  PROC DrawPart13()
    MoveL Offs(pOrigin,108.13,133.18,0.00),v40,z0,tPen\WObj:=wPaper;
    MoveL Offs(pOrigin,107.17,132.22,0.00),v40,z0,tPen\WObj:=wPaper;
    MoveL Offs(pOrigin,106.24,132.34,0.00),v40,z0,tPen\WObj:=wPaper;
    MoveL Offs(pOrigin,132.55,106.03,0.00),v40,z0,tPen\WObj:=wPaper;
    MoveL Offs(pOrigin,132.03,106.30,0.00),v40,z0,tPen\WObj:=wPaper;
    MoveL Offs(pOrigin,118.67,92.94,0.00),v40,z0,tPen\WObj:=wPaper;
    MoveL Offs(pOrigin,118.15,92.06,0.00),v40,z0,tPen\WObj:=wPaper;
    MoveL Offs(pOrigin,106.16,104.04,0.00),v40,z0,tPen\WObj:=wPaper;
    MoveL Offs(pOrigin,106.93,103.61,0.00),v40,z0,tPen\WObj:=wPaper;
    MoveL Offs(pOrigin,132.39,129.07,0.00),v40,z0,tPen\WObj:=wPaper;
    MoveL Offs(pOrigin,131.45,128.70,0.00),v40,z0,tPen\WObj:=wPaper;
    MoveL Offs(pOrigin,107.90,128.70,0.00),v40,z0,tPen\WObj:=wPaper;
    MoveL Offs(pOrigin,106.97,129.03,0.00),v40,z0,tPen\WObj:=wPaper;
    MoveL Offs(pOrigin,111.11,133.17,0.00),v40,fine,tPen\WObj:=wPaper;
    MoveL Offs(pOrigin,111.11,133.17,6.00),v60,z5,tPen\WObj:=wPaper;
    MoveL Offs(pOrigin,110.40,134.16,6.00),vTravel,z5,tPen\WObj:=wPaper;
    MoveL Offs(pOrigin,110.40,134.16,0.00),v60,z0,tPen\WObj:=wPaper;
    MoveL Offs(pOrigin,132.46,112.10,0.00),v40,z0,tPen\WObj:=wPaper;
    MoveL Offs(pOrigin,131.80,112.05,0.00),v40,z0,tPen\WObj:=wPaper;
    MoveL Offs(pOrigin,112.71,92.96,0.00),v40,z0,tPen\WObj:=wPaper;
    MoveL Offs(pOrigin,112.30,91.93,0.00),v40,z0,tPen\WObj:=wPaper;
    MoveL Offs(pOrigin,106.25,97.98,0.00),v40,z0,tPen\WObj:=wPaper;
    MoveL Offs(pOrigin,106.95,97.65,0.00),v40,z0,tPen\WObj:=wPaper;
    MoveL Offs(pOrigin,132.20,122.90,0.00),v40,z0,tPen\WObj:=wPaper;
    MoveL Offs(pOrigin,131.30,123.42,0.00),v40,z0,tPen\WObj:=wPaper;
    MoveL Offs(pOrigin,107.90,123.42,0.00),v40,z0,tPen\WObj:=wPaper;
    MoveL Offs(pOrigin,107.90,124.47,0.00),v40,z0,tPen\WObj:=wPaper;
    MoveL Offs(pOrigin,131.30,124.47,0.00),v40,z0,tPen\WObj:=wPaper;
    MoveL Offs(pOrigin,132.09,124.28,0.00),v40,z0,tPen\WObj:=wPaper;
    MoveL Offs(pOrigin,106.95,99.14,0.00),v40,z0,tPen\WObj:=wPaper;
    MoveL Offs(pOrigin,107.75,99.13,0.00),v40,z0,tPen\WObj:=wPaper;
    MoveL Offs(pOrigin,131.45,99.13,0.00),v40,z0,tPen\WObj:=wPaper;
    MoveL Offs(pOrigin,132.05,98.86,0.00),v40,z0,tPen\WObj:=wPaper;
    MoveL Offs(pOrigin,126.32,93.13,0.00),v40,z0,tPen\WObj:=wPaper;
    MoveL Offs(pOrigin,126.87,92.30,0.00),v40,z0,tPen\WObj:=wPaper;
    MoveL Offs(pOrigin,106.08,113.08,0.00),v40,z0,tPen\WObj:=wPaper;
    MoveL Offs(pOrigin,106.91,112.55,0.00),v40,z0,tPen\WObj:=wPaper;
    MoveL Offs(pOrigin,127.70,133.33,0.00),v40,z0,tPen\WObj:=wPaper;
    MoveL Offs(pOrigin,126.99,133.99,0.00),v40,z0,tPen\WObj:=wPaper;
    MoveL Offs(pOrigin,155.31,105.67,0.00),v40,z0,tPen\WObj:=wPaper;
    MoveL Offs(pOrigin,155.95,106.53,0.00),v40,z0,tPen\WObj:=wPaper;
    MoveL Offs(pOrigin,128.27,134.21,0.00),v40,fine,tPen\WObj:=wPaper;
    MoveL Offs(pOrigin,128.27,134.21,6.00),v60,z5,tPen\WObj:=wPaper;
    MoveL Offs(pOrigin,129.19,133.33,6.00),vTravel,z5,tPen\WObj:=wPaper;
    MoveL Offs(pOrigin,129.19,133.33,0.00),v60,z0,tPen\WObj:=wPaper;
    MoveL Offs(pOrigin,106.91,111.06,0.00),v40,z0,tPen\WObj:=wPaper;
    MoveL Offs(pOrigin,106.18,111.49,0.00),v40,z0,tPen\WObj:=wPaper;
    MoveL Offs(pOrigin,125.38,92.29,0.00),v40,z0,tPen\WObj:=wPaper;
    MoveL Offs(pOrigin,124.62,92.92,0.00),v40,z0,tPen\WObj:=wPaper;
    MoveL Offs(pOrigin,132.15,100.45,0.00),v40,z0,tPen\WObj:=wPaper;
    MoveL Offs(pOrigin,131.45,100.18,0.00),v40,z0,tPen\WObj:=wPaper;
    MoveL Offs(pOrigin,107.75,100.18,0.00),v40,z0,tPen\WObj:=wPaper;
    MoveL Offs(pOrigin,106.84,100.53,0.00),v40,z0,tPen\WObj:=wPaper;
    MoveL Offs(pOrigin,132.08,125.77,0.00),v40,z0,tPen\WObj:=wPaper;
    MoveL Offs(pOrigin,131.30,125.53,0.00),v40,z0,tPen\WObj:=wPaper;
    MoveL Offs(pOrigin,107.90,125.53,0.00),v40,z0,tPen\WObj:=wPaper;
    MoveL Offs(pOrigin,107.90,126.58,0.00),v40,z0,tPen\WObj:=wPaper;
    MoveL Offs(pOrigin,131.30,126.58,0.00),v40,z0,tPen\WObj:=wPaper;
    MoveL Offs(pOrigin,131.45,127.64,0.00),v40,z0,tPen\WObj:=wPaper;
    MoveL Offs(pOrigin,107.90,127.64,0.00),v40,z0,tPen\WObj:=wPaper;
    MoveL Offs(pOrigin,106.87,127.44,0.00),v40,z0,tPen\WObj:=wPaper;
    MoveL Offs(pOrigin,112.70,133.27,0.00),v40,z0,tPen\WObj:=wPaper;
    MoveL Offs(pOrigin,112.10,133.95,0.00),v40,z0,tPen\WObj:=wPaper;
    MoveL Offs(pOrigin,132.57,113.48,0.00),v40,z0,tPen\WObj:=wPaper;
    MoveL Offs(pOrigin,131.80,113.54,0.00),v40,z0,tPen\WObj:=wPaper;
    MoveL Offs(pOrigin,111.22,92.96,0.00),v40,z0,tPen\WObj:=wPaper;
    MoveL Offs(pOrigin,110.81,91.93,0.00),v40,z0,tPen\WObj:=wPaper;
    MoveL Offs(pOrigin,106.14,96.60,0.00),v40,z0,tPen\WObj:=wPaper;
    MoveL Offs(pOrigin,106.96,96.16,0.00),v40,z0,tPen\WObj:=wPaper;
    MoveL Offs(pOrigin,132.09,121.30,0.00),v40,z0,tPen\WObj:=wPaper;
    MoveL Offs(pOrigin,131.30,121.30,0.00),v40,z0,tPen\WObj:=wPaper;
    MoveL Offs(pOrigin,107.90,121.30,0.00),v40,z0,tPen\WObj:=wPaper;
    MoveL Offs(pOrigin,106.88,121.48,0.00),v40,z0,tPen\WObj:=wPaper;
    MoveL Offs(pOrigin,118.66,133.25,0.00),v40,z0,tPen\WObj:=wPaper;
    MoveL Offs(pOrigin,118.05,133.97,0.00),v40,z0,tPen\WObj:=wPaper;
    MoveL Offs(pOrigin,132.59,119.44,0.00),v40,z0,tPen\WObj:=wPaper;
    MoveL Offs(pOrigin,132.10,119.81,0.00),v40,z0,tPen\WObj:=wPaper;
    MoveL Offs(pOrigin,106.96,94.68,0.00),v40,z0,tPen\WObj:=wPaper;
    MoveL Offs(pOrigin,107.75,94.90,0.00),v40,z0,tPen\WObj:=wPaper;
    MoveL Offs(pOrigin,131.30,94.90,0.00),v40,z0,tPen\WObj:=wPaper;
    MoveL Offs(pOrigin,132.06,94.39,0.00),v40,z0,tPen\WObj:=wPaper;
    MoveL Offs(pOrigin,130.79,93.12,0.00),v40,z0,tPen\WObj:=wPaper;
    MoveL Offs(pOrigin,131.00,93.85,0.00),v40,z0,tPen\WObj:=wPaper;
    MoveL Offs(pOrigin,108.05,93.85,0.00),v40,z0,tPen\WObj:=wPaper;
    MoveL Offs(pOrigin,107.28,93.50,0.00),v40,z0,tPen\WObj:=wPaper;
    MoveL Offs(pOrigin,131.89,118.11,0.00),v40,z0,tPen\WObj:=wPaper;
    MoveL Offs(pOrigin,132.58,117.95,0.00),v40,z0,tPen\WObj:=wPaper;
    MoveL Offs(pOrigin,116.35,134.17,0.00),v40,z0,tPen\WObj:=wPaper;
    MoveL Offs(pOrigin,115.78,133.37,0.00),v40,z0,tPen\WObj:=wPaper;
    MoveL Offs(pOrigin,106.88,124.46,0.00),v40,z0,tPen\WObj:=wPaper;
    MoveL Offs(pOrigin,106.22,124.89,0.00),v40,z0,tPen\WObj:=wPaper;
    MoveL Offs(pOrigin,132.63,98.48,0.00),v40,fine,tPen\WObj:=wPaper;
    MoveL Offs(pOrigin,132.63,98.48,6.00),v60,z5,tPen\WObj:=wPaper;
    MoveL Offs(pOrigin,131.45,98.07,6.00),vTravel,z5,tPen\WObj:=wPaper;
    MoveL Offs(pOrigin,131.45,98.07,0.00),v60,z0,tPen\WObj:=wPaper;
    MoveL Offs(pOrigin,107.75,98.07,0.00),v40,z0,tPen\WObj:=wPaper;
    MoveL Offs(pOrigin,107.75,97.02,0.00),v40,z0,tPen\WObj:=wPaper;
    MoveL Offs(pOrigin,131.45,97.02,0.00),v40,z0,tPen\WObj:=wPaper;
    MoveL Offs(pOrigin,132.06,97.37,0.00),v40,z0,tPen\WObj:=wPaper;
    MoveL Offs(pOrigin,127.81,93.13,0.00),v40,z0,tPen\WObj:=wPaper;
    MoveL Offs(pOrigin,128.36,92.30,0.00),v40,z0,tPen\WObj:=wPaper;
    MoveL Offs(pOrigin,105.56,115.10,0.00),v40,fine,tPen\WObj:=wPaper;
    MoveL Offs(pOrigin,105.56,115.10,6.00),v60,z5,tPen\WObj:=wPaper;
    MoveL Offs(pOrigin,105.88,116.27,6.00),vTravel,z5,tPen\WObj:=wPaper;
    MoveL Offs(pOrigin,105.88,116.27,0.00),v60,z0,tPen\WObj:=wPaper;
    MoveL Offs(pOrigin,129.96,92.20,0.00),v40,z0,tPen\WObj:=wPaper;
    MoveL Offs(pOrigin,129.42,91.24,0.00),v40,z0,tPen\WObj:=wPaper;
    MoveL Offs(pOrigin,132.81,87.84,0.00),v40,fine,tPen\WObj:=wPaper;
    MoveL Offs(pOrigin,132.81,87.84,6.00),v60,z5,tPen\WObj:=wPaper;
    MoveL Offs(pOrigin,133.99,88.17,6.00),vTravel,z5,tPen\WObj:=wPaper;
    MoveL Offs(pOrigin,133.99,88.17,0.00),v60,z0,tPen\WObj:=wPaper;
    MoveL Offs(pOrigin,160.82,61.33,0.00),v40,z0,tPen\WObj:=wPaper;
    MoveL Offs(pOrigin,159.95,61.12,0.00),v40,z0,tPen\WObj:=wPaper;
    MoveL Offs(pOrigin,157.55,58.28,0.00),v40,z0,tPen\WObj:=wPaper;
    MoveL Offs(pOrigin,154.55,55.72,0.00),v40,z0,tPen\WObj:=wPaper;
    MoveL Offs(pOrigin,149.00,52.62,0.00),v40,z0,tPen\WObj:=wPaper;
    MoveL Offs(pOrigin,145.10,51.38,0.00),v40,z0,tPen\WObj:=wPaper;
    MoveL Offs(pOrigin,140.75,50.62,0.00),v40,z0,tPen\WObj:=wPaper;
    MoveL Offs(pOrigin,134.65,50.83,0.00),v40,z0,tPen\WObj:=wPaper;
    MoveL Offs(pOrigin,134.65,90.47,0.00),v40,z0,tPen\WObj:=wPaper;
  ENDPROC

  PROC DrawPart14()
    MoveL Offs(pOrigin,161.75,90.47,0.00),v40,z0,tPen\WObj:=wPaper;
    MoveL Offs(pOrigin,163.30,87.53,0.00),v40,z0,tPen\WObj:=wPaper;
    MoveL Offs(pOrigin,164.60,83.32,0.00),v40,z0,tPen\WObj:=wPaper;
    MoveL Offs(pOrigin,165.05,80.62,0.00),v40,z0,tPen\WObj:=wPaper;
    MoveL Offs(pOrigin,165.05,74.32,0.00),v40,z0,tPen\WObj:=wPaper;
    MoveL Offs(pOrigin,164.60,71.62,0.00),v40,z0,tPen\WObj:=wPaper;
    MoveL Offs(pOrigin,163.30,67.28,0.00),v40,z0,tPen\WObj:=wPaper;
    MoveL Offs(pOrigin,161.70,63.83,0.00),v40,z0,tPen\WObj:=wPaper;
    MoveL Offs(pOrigin,159.95,61.12,0.00),v40,z0,tPen\WObj:=wPaper;
    MoveL Offs(pOrigin,160.29,60.37,0.00),v40,z0,tPen\WObj:=wPaper;
    MoveL Offs(pOrigin,133.98,86.68,0.00),v40,z0,tPen\WObj:=wPaper;
    MoveL Offs(pOrigin,134.85,86.72,0.00),v40,z0,tPen\WObj:=wPaper;
    MoveL Offs(pOrigin,138.35,90.22,0.00),v40,z0,tPen\WObj:=wPaper;
    MoveL Offs(pOrigin,138.78,90.84,0.00),v40,z0,tPen\WObj:=wPaper;
    MoveL Offs(pOrigin,163.39,66.23,0.00),v40,z0,tPen\WObj:=wPaper;
    MoveL Offs(pOrigin,162.88,66.97,0.00),v40,z0,tPen\WObj:=wPaper;
    MoveL Offs(pOrigin,148.56,52.65,0.00),v40,z0,tPen\WObj:=wPaper;
    MoveL Offs(pOrigin,149.20,52.05,0.00),v40,z0,tPen\WObj:=wPaper;
    MoveL Offs(pOrigin,134.03,67.21,0.00),v40,z0,tPen\WObj:=wPaper;
    MoveL Offs(pOrigin,134.80,67.26,0.00),v40,z0,tPen\WObj:=wPaper;
    MoveL Offs(pOrigin,158.14,90.59,0.00),v40,fine,tPen\WObj:=wPaper;
    MoveL Offs(pOrigin,158.14,90.59,6.00),v60,z5,tPen\WObj:=wPaper;
    MoveL Offs(pOrigin,159.31,91.22,6.00),vTravel,z5,tPen\WObj:=wPaper;
    MoveL Offs(pOrigin,159.31,91.22,0.00),v60,z0,tPen\WObj:=wPaper;
    MoveL Offs(pOrigin,164.40,86.13,0.00),v40,z0,tPen\WObj:=wPaper;
    MoveL Offs(pOrigin,163.79,85.79,0.00),v40,z0,tPen\WObj:=wPaper;
    MoveL Offs(pOrigin,134.72,56.73,0.00),v40,z0,tPen\WObj:=wPaper;
    MoveL Offs(pOrigin,134.00,56.79,0.00),v40,z0,tPen\WObj:=wPaper;
    MoveL Offs(pOrigin,140.79,50.00,0.00),v40,z0,tPen\WObj:=wPaper;
    MoveL Offs(pOrigin,140.70,50.76,0.00),v40,z0,tPen\WObj:=wPaper;
    MoveL Offs(pOrigin,164.88,74.94,0.00),v40,z0,tPen\WObj:=wPaper;
    MoveL Offs(pOrigin,164.15,74.84,0.00),v40,z0,tPen\WObj:=wPaper;
    MoveL Offs(pOrigin,135.80,74.84,0.00),v40,z0,tPen\WObj:=wPaper;
    MoveL Offs(pOrigin,134.78,74.71,0.00),v40,z0,tPen\WObj:=wPaper;
    MoveL Offs(pOrigin,150.58,90.51,0.00),v40,z0,tPen\WObj:=wPaper;
    MoveL Offs(pOrigin,150.38,91.19,0.00),v40,z0,tPen\WObj:=wPaper;
    MoveL Offs(pOrigin,165.86,75.71,0.00),v40,fine,tPen\WObj:=wPaper;
    MoveL Offs(pOrigin,165.86,75.71,6.00),v60,z5,tPen\WObj:=wPaper;
    MoveL Offs(pOrigin,165.09,76.64,6.00),vTravel,z5,tPen\WObj:=wPaper;
    MoveL Offs(pOrigin,165.09,76.64,0.00),v60,z0,tPen\WObj:=wPaper;
    MoveL Offs(pOrigin,139.21,50.76,0.00),v40,z0,tPen\WObj:=wPaper;
    MoveL Offs(pOrigin,139.41,49.89,0.00),v40,z0,tPen\WObj:=wPaper;
    MoveL Offs(pOrigin,134.00,55.30,0.00),v40,z0,tPen\WObj:=wPaper;
    MoveL Offs(pOrigin,134.73,55.24,0.00),v40,z0,tPen\WObj:=wPaper;
    MoveL Offs(pOrigin,164.11,84.62,0.00),v40,z0,tPen\WObj:=wPaper;
    MoveL Offs(pOrigin,163.40,84.34,0.00),v40,z0,tPen\WObj:=wPaper;
    MoveL Offs(pOrigin,135.80,84.34,0.00),v40,z0,tPen\WObj:=wPaper;
    MoveL Offs(pOrigin,135.80,85.40,0.00),v40,z0,tPen\WObj:=wPaper;
    MoveL Offs(pOrigin,163.10,85.40,0.00),v40,z0,tPen\WObj:=wPaper;
    MoveL Offs(pOrigin,162.65,86.46,0.00),v40,z0,tPen\WObj:=wPaper;
    MoveL Offs(pOrigin,135.80,86.46,0.00),v40,z0,tPen\WObj:=wPaper;
    MoveL Offs(pOrigin,135.65,87.51,0.00),v40,z0,tPen\WObj:=wPaper;
    MoveL Offs(pOrigin,162.20,87.51,0.00),v40,z0,tPen\WObj:=wPaper;
    MoveL Offs(pOrigin,162.93,87.92,0.00),v40,z0,tPen\WObj:=wPaper;
    MoveL Offs(pOrigin,134.72,59.71,0.00),v40,z0,tPen\WObj:=wPaper;
    MoveL Offs(pOrigin,133.80,59.98,0.00),v40,z0,tPen\WObj:=wPaper;
    MoveL Offs(pOrigin,143.66,50.11,0.00),v40,fine,tPen\WObj:=wPaper;
    MoveL Offs(pOrigin,143.66,50.11,6.00),v60,z5,tPen\WObj:=wPaper;
    MoveL Offs(pOrigin,144.83,50.44,6.00),vTravel,z5,tPen\WObj:=wPaper;
    MoveL Offs(pOrigin,144.83,50.44,0.00),v60,z0,tPen\WObj:=wPaper;
    MoveL Offs(pOrigin,134.12,61.15,0.00),v40,z0,tPen\WObj:=wPaper;
    MoveL Offs(pOrigin,134.71,61.20,0.00),v40,z0,tPen\WObj:=wPaper;
    MoveL Offs(pOrigin,162.50,88.99,0.00),v40,z0,tPen\WObj:=wPaper;
    MoveL Offs(pOrigin,161.75,88.57,0.00),v40,z0,tPen\WObj:=wPaper;
    MoveL Offs(pOrigin,135.65,88.57,0.00),v40,z0,tPen\WObj:=wPaper;
    MoveL Offs(pOrigin,134.74,88.11,0.00),v40,z0,tPen\WObj:=wPaper;
    MoveL Offs(pOrigin,137.07,90.44,0.00),v40,z0,tPen\WObj:=wPaper;
    MoveL Offs(pOrigin,136.97,91.15,0.00),v40,z0,tPen\WObj:=wPaper;
    MoveL Offs(pOrigin,162.96,65.17,0.00),v40,z0,tPen\WObj:=wPaper;
    MoveL Offs(pOrigin,162.53,64.10,0.00),v40,z0,tPen\WObj:=wPaper;
    MoveL Offs(pOrigin,135.70,90.94,0.00),v40,z0,tPen\WObj:=wPaper;
    MoveL Offs(pOrigin,134.74,90.40,0.00),v40,z0,tPen\WObj:=wPaper;
    MoveL Offs(pOrigin,161.89,63.25,0.00),v40,z0,tPen\WObj:=wPaper;
    MoveL Offs(pOrigin,161.25,62.40,0.00),v40,z0,tPen\WObj:=wPaper;
    MoveL Offs(pOrigin,134.20,89.44,0.00),v40,fine,tPen\WObj:=wPaper;
    MoveL Offs(pOrigin,134.20,89.44,6.00),v60,z5,tPen\WObj:=wPaper;
    MoveL Offs(pOrigin,132.15,90.47,6.00),vTravel,z5,tPen\WObj:=wPaper;
    MoveL Offs(pOrigin,132.15,90.47,0.00),v60,z0,tPen\WObj:=wPaper;
    MoveL Offs(pOrigin,107.30,90.47,0.00),v40,z0,tPen\WObj:=wPaper;
    MoveL Offs(pOrigin,107.00,90.07,0.00),v40,z0,tPen\WObj:=wPaper;
    MoveL Offs(pOrigin,107.05,50.92,0.00),v40,z0,tPen\WObj:=wPaper;
    MoveL Offs(pOrigin,110.60,50.62,0.00),v40,z0,tPen\WObj:=wPaper;
    MoveL Offs(pOrigin,131.90,50.67,0.00),v40,z0,tPen\WObj:=wPaper;
    MoveL Offs(pOrigin,132.20,51.08,0.00),v40,z0,tPen\WObj:=wPaper;
    MoveL Offs(pOrigin,132.15,90.47,0.00),v40,fine,tPen\WObj:=wPaper;
    MoveL Offs(pOrigin,132.15,90.47,6.00),v60,z5,tPen\WObj:=wPaper;
    MoveL Offs(pOrigin,130.55,89.62,6.00),vTravel,z5,tPen\WObj:=wPaper;
    MoveL Offs(pOrigin,130.55,89.62,0.00),v60,z0,tPen\WObj:=wPaper;
    MoveL Offs(pOrigin,127.40,89.62,0.00),v40,z0,tPen\WObj:=wPaper;
    MoveL Offs(pOrigin,128.14,90.47,0.00),v40,z0,tPen\WObj:=wPaper;
    MoveL Offs(pOrigin,106.93,69.25,0.00),v40,z0,tPen\WObj:=wPaper;
    MoveL Offs(pOrigin,106.17,69.69,0.00),v40,z0,tPen\WObj:=wPaper;
    MoveL Offs(pOrigin,126.01,49.85,0.00),v40,z0,tPen\WObj:=wPaper;
    MoveL Offs(pOrigin,125.81,50.80,0.00),v40,z0,tPen\WObj:=wPaper;
    MoveL Offs(pOrigin,132.06,57.06,0.00),v40,z0,tPen\WObj:=wPaper;
    MoveL Offs(pOrigin,131.30,56.89,0.00),v40,z0,tPen\WObj:=wPaper;
    MoveL Offs(pOrigin,107.90,56.89,0.00),v40,z0,tPen\WObj:=wPaper;
    MoveL Offs(pOrigin,106.96,57.34,0.00),v40,z0,tPen\WObj:=wPaper;
    MoveL Offs(pOrigin,131.89,82.27,0.00),v40,z0,tPen\WObj:=wPaper;
    MoveL Offs(pOrigin,132.48,82.21,0.00),v40,z0,tPen\WObj:=wPaper;
    MoveL Offs(pOrigin,105.75,108.93,0.00),v40,fine,tPen\WObj:=wPaper;
    MoveL Offs(pOrigin,105.75,108.93,6.00),v60,z5,tPen\WObj:=wPaper;
    MoveL Offs(pOrigin,106.07,110.11,6.00),vTravel,z5,tPen\WObj:=wPaper;
    MoveL Offs(pOrigin,106.07,110.11,0.00),v60,z0,tPen\WObj:=wPaper;
    MoveL Offs(pOrigin,124.10,92.07,0.00),v40,fine,tPen\WObj:=wPaper;
    MoveL Offs(pOrigin,124.10,92.07,6.00),v60,z5,tPen\WObj:=wPaper;
    MoveL Offs(pOrigin,123.13,92.93,6.00),vTravel,z5,tPen\WObj:=wPaper;
    MoveL Offs(pOrigin,123.13,92.93,0.00),v60,z0,tPen\WObj:=wPaper;
    MoveL Offs(pOrigin,132.15,101.94,0.00),v40,z0,tPen\WObj:=wPaper;
    MoveL Offs(pOrigin,131.45,102.30,0.00),v40,z0,tPen\WObj:=wPaper;
    MoveL Offs(pOrigin,107.75,102.30,0.00),v40,z0,tPen\WObj:=wPaper;
    MoveL Offs(pOrigin,106.83,102.02,0.00),v40,z0,tPen\WObj:=wPaper;
    MoveL Offs(pOrigin,132.18,127.36,0.00),v40,z0,tPen\WObj:=wPaper;
    MoveL Offs(pOrigin,132.82,126.67,0.00),v40,z0,tPen\WObj:=wPaper;
    MoveL Offs(pOrigin,125.50,133.99,0.00),v40,z0,tPen\WObj:=wPaper;
    MoveL Offs(pOrigin,126.10,133.23,0.00),v40,z0,tPen\WObj:=wPaper;
    MoveL Offs(pOrigin,106.91,114.03,0.00),v40,z0,tPen\WObj:=wPaper;
    MoveL Offs(pOrigin,107.90,113.91,0.00),v40,z0,tPen\WObj:=wPaper;
    MoveL Offs(pOrigin,131.00,113.91,0.00),v40,z0,tPen\WObj:=wPaper;
    MoveL Offs(pOrigin,131.00,114.97,0.00),v40,z0,tPen\WObj:=wPaper;
  ENDPROC

  PROC DrawPart15()
    MoveL Offs(pOrigin,108.05,114.97,0.00),v40,z0,tPen\WObj:=wPaper;
    MoveL Offs(pOrigin,107.90,116.02,0.00),v40,z0,tPen\WObj:=wPaper;
    MoveL Offs(pOrigin,131.15,116.02,0.00),v40,z0,tPen\WObj:=wPaper;
    MoveL Offs(pOrigin,131.15,117.08,0.00),v40,z0,tPen\WObj:=wPaper;
    MoveL Offs(pOrigin,107.90,117.08,0.00),v40,z0,tPen\WObj:=wPaper;
    MoveL Offs(pOrigin,106.90,117.01,0.00),v40,z0,tPen\WObj:=wPaper;
    MoveL Offs(pOrigin,123.23,133.35,0.00),v40,z0,tPen\WObj:=wPaper;
    MoveL Offs(pOrigin,123.80,134.20,0.00),v40,z0,tPen\WObj:=wPaper;
    MoveL Offs(pOrigin,132.81,125.18,0.00),v40,fine,tPen\WObj:=wPaper;
    MoveL Offs(pOrigin,132.81,125.18,6.00),v60,z5,tPen\WObj:=wPaper;
    MoveL Offs(pOrigin,133.99,125.50,6.00),vTravel,z5,tPen\WObj:=wPaper;
    MoveL Offs(pOrigin,133.99,125.50,0.00),v60,z0,tPen\WObj:=wPaper;
    MoveL Offs(pOrigin,154.67,104.82,0.00),v40,z0,tPen\WObj:=wPaper;
    MoveL Offs(pOrigin,154.25,105.07,0.00),v40,z0,tPen\WObj:=wPaper;
    MoveL Offs(pOrigin,156.25,108.18,0.00),v40,z0,tPen\WObj:=wPaper;
    MoveL Offs(pOrigin,152.05,102.78,0.00),v40,z0,tPen\WObj:=wPaper;
    MoveL Offs(pOrigin,154.25,105.07,0.00),v40,z0,tPen\WObj:=wPaper;
    MoveL Offs(pOrigin,153.50,105.46,0.00),v40,z0,tPen\WObj:=wPaper;
    MoveL Offs(pOrigin,135.65,105.46,0.00),v40,z0,tPen\WObj:=wPaper;
    MoveL Offs(pOrigin,134.80,106.08,0.00),v40,z0,tPen\WObj:=wPaper;
    MoveL Offs(pOrigin,154.42,125.71,0.00),v40,z0,tPen\WObj:=wPaper;
    MoveL Offs(pOrigin,153.65,125.53,0.00),v40,z0,tPen\WObj:=wPaper;
    MoveL Offs(pOrigin,135.50,125.53,0.00),v40,z0,tPen\WObj:=wPaper;
    MoveL Offs(pOrigin,134.74,125.44,0.00),v40,z0,tPen\WObj:=wPaper;
    MoveL Offs(pOrigin,142.48,133.19,0.00),v40,z0,tPen\WObj:=wPaper;
    MoveL Offs(pOrigin,141.99,133.93,0.00),v40,z0,tPen\WObj:=wPaper;
    MoveL Offs(pOrigin,158.43,117.49,0.00),v40,z0,tPen\WObj:=wPaper;
    MoveL Offs(pOrigin,157.74,117.08,0.00),v40,z0,tPen\WObj:=wPaper;
    MoveL Offs(pOrigin,134.72,94.06,0.00),v40,z0,tPen\WObj:=wPaper;
    MoveL Offs(pOrigin,134.60,93.53,0.00),v40,z0,tPen\WObj:=wPaper;
    MoveL Offs(pOrigin,134.60,98.18,0.00),v40,z0,tPen\WObj:=wPaper;
    MoveL Offs(pOrigin,134.60,93.53,0.00),v40,z0,tPen\WObj:=wPaper;
    MoveL Offs(pOrigin,135.05,92.93,0.00),v40,z0,tPen\WObj:=wPaper;
    MoveL Offs(pOrigin,136.25,92.93,0.00),v40,z0,tPen\WObj:=wPaper;
    MoveL Offs(pOrigin,135.05,92.93,0.00),v40,z0,tPen\WObj:=wPaper;
    MoveL Offs(pOrigin,135.36,93.21,0.00),v40,z0,tPen\WObj:=wPaper;
    MoveL Offs(pOrigin,157.53,115.38,0.00),v40,z0,tPen\WObj:=wPaper;
    MoveL Offs(pOrigin,158.21,114.72,0.00),v40,z0,tPen\WObj:=wPaper;
    MoveL Offs(pOrigin,139.01,133.92,0.00),v40,z0,tPen\WObj:=wPaper;
    MoveL Offs(pOrigin,139.61,133.30,0.00),v40,z0,tPen\WObj:=wPaper;
    MoveL Offs(pOrigin,134.52,128.21,0.00),v40,z0,tPen\WObj:=wPaper;
    MoveL Offs(pOrigin,135.35,128.70,0.00),v40,z0,tPen\WObj:=wPaper;
    MoveL Offs(pOrigin,150.65,128.70,0.00),v40,z0,tPen\WObj:=wPaper;
    MoveL Offs(pOrigin,150.90,129.65,0.00),v40,z0,tPen\WObj:=wPaper;
    MoveL Offs(pOrigin,134.78,113.53,0.00),v40,z0,tPen\WObj:=wPaper;
    MoveL Offs(pOrigin,134.06,113.48,0.00),v40,z0,tPen\WObj:=wPaper;
    MoveL Offs(pOrigin,155.27,92.27,0.00),v40,z0,tPen\WObj:=wPaper;
    MoveL Offs(pOrigin,156.00,92.94,0.00),v40,z0,tPen\WObj:=wPaper;
    MoveL Offs(pOrigin,158.23,95.17,0.00),v40,z0,tPen\WObj:=wPaper;
    MoveL Offs(pOrigin,157.25,94.90,0.00),v40,z0,tPen\WObj:=wPaper;
    MoveL Offs(pOrigin,135.35,94.90,0.00),v40,z0,tPen\WObj:=wPaper;
    MoveL Offs(pOrigin,134.72,95.55,0.00),v40,z0,tPen\WObj:=wPaper;
    MoveL Offs(pOrigin,157.52,118.36,0.00),v40,z0,tPen\WObj:=wPaper;
    MoveL Offs(pOrigin,157.55,119.18,0.00),v40,z0,tPen\WObj:=wPaper;
    MoveL Offs(pOrigin,156.30,122.93,0.00),v40,z0,tPen\WObj:=wPaper;
    MoveL Offs(pOrigin,153.45,127.28,0.00),v40,z0,tPen\WObj:=wPaper;
    MoveL Offs(pOrigin,149.50,130.62,0.00),v40,z0,tPen\WObj:=wPaper;
    MoveL Offs(pOrigin,157.25,111.22,0.00),v40,z0,tPen\WObj:=wPaper;
    MoveL Offs(pOrigin,157.70,113.03,0.00),v40,z0,tPen\WObj:=wPaper;
    MoveL Offs(pOrigin,157.85,116.47,0.00),v40,z0,tPen\WObj:=wPaper;
    MoveL Offs(pOrigin,157.55,119.18,0.00),v40,z0,tPen\WObj:=wPaper;
    MoveL Offs(pOrigin,157.20,119.53,0.00),v40,z0,tPen\WObj:=wPaper;
    MoveL Offs(pOrigin,134.72,97.04,0.00),v40,z0,tPen\WObj:=wPaper;
    MoveL Offs(pOrigin,134.12,97.00,0.00),v40,z0,tPen\WObj:=wPaper;
    MoveL Offs(pOrigin,138.68,92.44,0.00),v40,z0,tPen\WObj:=wPaper;
    MoveL Offs(pOrigin,138.24,93.10,0.00),v40,z0,tPen\WObj:=wPaper;
    MoveL Offs(pOrigin,157.43,112.30,0.00),v40,z0,tPen\WObj:=wPaper;
    MoveL Offs(pOrigin,158.20,111.74,0.00),v40,z0,tPen\WObj:=wPaper;
    MoveL Offs(pOrigin,135.71,134.23,0.00),v40,z0,tPen\WObj:=wPaper;
    MoveL Offs(pOrigin,135.20,133.27,0.00),v40,z0,tPen\WObj:=wPaper;
    MoveL Offs(pOrigin,141.35,133.27,0.00),v40,z0,tPen\WObj:=wPaper;
    MoveL Offs(pOrigin,143.60,132.98,0.00),v40,z0,tPen\WObj:=wPaper;
    MoveL Offs(pOrigin,147.50,131.73,0.00),v40,z0,tPen\WObj:=wPaper;
    MoveL Offs(pOrigin,149.20,130.77,0.00),v40,z0,tPen\WObj:=wPaper;
    MoveL Offs(pOrigin,134.60,130.57,0.00),v40,z0,tPen\WObj:=wPaper;
    MoveL Offs(pOrigin,134.60,132.98,0.00),v40,z0,tPen\WObj:=wPaper;
    MoveL Offs(pOrigin,135.20,133.27,0.00),v40,z0,tPen\WObj:=wPaper;
    MoveL Offs(pOrigin,134.75,133.69,0.00),v40,z0,tPen\WObj:=wPaper;
    MoveL Offs(pOrigin,157.88,110.57,0.00),v40,z0,tPen\WObj:=wPaper;
    MoveL Offs(pOrigin,156.91,110.28,0.00),v40,z0,tPen\WObj:=wPaper;
    MoveL Offs(pOrigin,139.73,93.09,0.00),v40,z0,tPen\WObj:=wPaper;
    MoveL Offs(pOrigin,140.17,92.44,0.00),v40,z0,tPen\WObj:=wPaper;
    MoveL Offs(pOrigin,134.12,98.49,0.00),v40,z0,tPen\WObj:=wPaper;
    MoveL Offs(pOrigin,134.60,98.62,0.00),v40,z0,tPen\WObj:=wPaper;
    MoveL Offs(pOrigin,134.60,110.03,0.00),v40,z0,tPen\WObj:=wPaper;
    MoveL Offs(pOrigin,134.60,98.62,0.00),v40,z0,tPen\WObj:=wPaper;
    MoveL Offs(pOrigin,134.71,98.53,0.00),v40,z0,tPen\WObj:=wPaper;
    MoveL Offs(pOrigin,156.88,120.70,0.00),v40,z0,tPen\WObj:=wPaper;
    MoveL Offs(pOrigin,156.20,120.25,0.00),v40,z0,tPen\WObj:=wPaper;
    MoveL Offs(pOrigin,135.65,120.25,0.00),v40,z0,tPen\WObj:=wPaper;
    MoveL Offs(pOrigin,134.86,119.59,0.00),v40,z0,tPen\WObj:=wPaper;
    MoveL Offs(pOrigin,147.06,131.79,0.00),v40,z0,tPen\WObj:=wPaper;
    MoveL Offs(pOrigin,147.35,130.81,0.00),v40,z0,tPen\WObj:=wPaper;
    MoveL Offs(pOrigin,135.35,130.81,0.00),v40,z0,tPen\WObj:=wPaper;
    MoveL Offs(pOrigin,134.41,131.08,0.00),v40,z0,tPen\WObj:=wPaper;
    MoveL Offs(pOrigin,136.63,133.31,0.00),v40,z0,tPen\WObj:=wPaper;
    MoveL Offs(pOrigin,137.31,134.13,0.00),v40,z0,tPen\WObj:=wPaper;
    MoveL Offs(pOrigin,158.20,113.23,0.00),v40,z0,tPen\WObj:=wPaper;
    MoveL Offs(pOrigin,157.54,113.89,0.00),v40,z0,tPen\WObj:=wPaper;
    MoveL Offs(pOrigin,136.75,93.10,0.00),v40,z0,tPen\WObj:=wPaper;
    MoveL Offs(pOrigin,136.55,92.93,0.00),v40,z0,tPen\WObj:=wPaper;
    MoveL Offs(pOrigin,159.50,92.93,0.00),v40,z0,tPen\WObj:=wPaper;
    MoveL Offs(pOrigin,159.80,93.38,0.00),v40,z0,tPen\WObj:=wPaper;
    MoveL Offs(pOrigin,156.80,96.62,0.00),v40,z0,tPen\WObj:=wPaper;
    MoveL Offs(pOrigin,154.60,98.38,0.00),v40,z0,tPen\WObj:=wPaper;
    MoveL Offs(pOrigin,136.55,92.93,0.00),v40,z0,tPen\WObj:=wPaper;
    MoveL Offs(pOrigin,137.30,92.32,0.00),v40,z0,tPen\WObj:=wPaper;
    MoveL Offs(pOrigin,134.01,95.61,0.00),v40,fine,tPen\WObj:=wPaper;
    MoveL Offs(pOrigin,134.01,95.61,6.00),v60,z5,tPen\WObj:=wPaper;
    MoveL Offs(pOrigin,132.84,95.29,6.00),vTravel,z5,tPen\WObj:=wPaper;
    MoveL Offs(pOrigin,132.84,95.29,0.00),v60,z0,tPen\WObj:=wPaper;
    MoveL Offs(pOrigin,105.58,122.55,0.00),v40,fine,tPen\WObj:=wPaper;
    MoveL Offs(pOrigin,105.58,122.55,6.00),v60,z5,tPen\WObj:=wPaper;
    MoveL Offs(pOrigin,105.90,123.72,6.00),vTravel,z5,tPen\WObj:=wPaper;
    MoveL Offs(pOrigin,105.90,123.72,0.00),v60,z0,tPen\WObj:=wPaper;
    MoveL Offs(pOrigin,132.63,96.99,0.00),v40,fine,tPen\WObj:=wPaper;
    MoveL Offs(pOrigin,132.63,96.99,6.00),v60,z5,tPen\WObj:=wPaper;
    MoveL Offs(pOrigin,132.06,95.88,6.00),vTravel,z5,tPen\WObj:=wPaper;
    MoveL Offs(pOrigin,132.06,95.88,0.00),v60,z0,tPen\WObj:=wPaper;
    MoveL Offs(pOrigin,129.30,93.12,0.00),v40,fine,tPen\WObj:=wPaper;
  ENDPROC

  PROC DrawPart16()
    MoveL Offs(pOrigin,129.30,93.12,6.00),v60,z5,tPen\WObj:=wPaper;
    MoveL Offs(pOrigin,128.31,94.87,6.00),vTravel,z5,tPen\WObj:=wPaper;
    MoveL Offs(pOrigin,128.31,94.87,0.00),v60,z0,tPen\WObj:=wPaper;
    MoveL Offs(pOrigin,128.31,105.82,0.00),v40,z0,tPen\WObj:=wPaper;
    MoveL Offs(pOrigin,127.26,105.82,0.00),v40,z0,tPen\WObj:=wPaper;
    MoveL Offs(pOrigin,127.26,94.72,0.00),v40,z0,tPen\WObj:=wPaper;
    MoveL Offs(pOrigin,126.20,94.72,0.00),v40,z0,tPen\WObj:=wPaper;
    MoveL Offs(pOrigin,126.20,105.52,0.00),v40,fine,tPen\WObj:=wPaper;
    MoveL Offs(pOrigin,126.20,105.52,6.00),v60,z5,tPen\WObj:=wPaper;
    MoveL Offs(pOrigin,125.14,104.32,6.00),vTravel,z5,tPen\WObj:=wPaper;
    MoveL Offs(pOrigin,125.14,104.32,0.00),v60,z0,tPen\WObj:=wPaper;
    MoveL Offs(pOrigin,125.14,94.72,0.00),v40,z0,tPen\WObj:=wPaper;
    MoveL Offs(pOrigin,124.09,94.72,0.00),v40,z0,tPen\WObj:=wPaper;
    MoveL Offs(pOrigin,124.09,103.58,0.00),v40,z0,tPen\WObj:=wPaper;
    MoveL Offs(pOrigin,123.03,103.12,0.00),v40,z0,tPen\WObj:=wPaper;
    MoveL Offs(pOrigin,123.03,94.72,0.00),v40,z0,tPen\WObj:=wPaper;
    MoveL Offs(pOrigin,121.98,94.72,0.00),v40,z0,tPen\WObj:=wPaper;
    MoveL Offs(pOrigin,121.98,102.08,0.00),v40,z0,tPen\WObj:=wPaper;
    MoveL Offs(pOrigin,120.92,101.78,0.00),v40,z0,tPen\WObj:=wPaper;
    MoveL Offs(pOrigin,120.92,97.28,0.00),v40,z0,tPen\WObj:=wPaper;
    MoveL Offs(pOrigin,119.86,97.57,0.00),v40,z0,tPen\WObj:=wPaper;
    MoveL Offs(pOrigin,119.86,102.38,0.00),v40,fine,tPen\WObj:=wPaper;
    MoveL Offs(pOrigin,119.86,102.38,6.00),v60,z5,tPen\WObj:=wPaper;
    MoveL Offs(pOrigin,118.81,103.28,6.00),vTravel,z5,tPen\WObj:=wPaper;
    MoveL Offs(pOrigin,118.81,103.28,0.00),v60,z0,tPen\WObj:=wPaper;
    MoveL Offs(pOrigin,118.81,97.72,0.00),v40,fine,tPen\WObj:=wPaper;
    MoveL Offs(pOrigin,118.81,97.72,6.00),v60,z5,tPen\WObj:=wPaper;
    MoveL Offs(pOrigin,117.75,96.67,6.00),vTravel,z5,tPen\WObj:=wPaper;
    MoveL Offs(pOrigin,117.75,96.67,0.00),v60,z0,tPen\WObj:=wPaper;
    MoveL Offs(pOrigin,117.75,105.98,0.00),v40,z0,tPen\WObj:=wPaper;
    MoveL Offs(pOrigin,118.81,105.98,0.00),v40,z0,tPen\WObj:=wPaper;
    MoveL Offs(pOrigin,118.81,104.62,0.00),v40,fine,tPen\WObj:=wPaper;
    MoveL Offs(pOrigin,118.81,104.62,6.00),v60,z5,tPen\WObj:=wPaper;
    MoveL Offs(pOrigin,116.70,105.98,6.00),vTravel,z5,tPen\WObj:=wPaper;
    MoveL Offs(pOrigin,116.70,105.98,0.00),v60,z0,tPen\WObj:=wPaper;
    MoveL Offs(pOrigin,116.70,95.78,0.00),v40,fine,tPen\WObj:=wPaper;
    MoveL Offs(pOrigin,116.70,95.78,6.00),v60,z5,tPen\WObj:=wPaper;
    MoveL Offs(pOrigin,115.64,95.02,6.00),vTravel,z5,tPen\WObj:=wPaper;
    MoveL Offs(pOrigin,115.64,95.02,0.00),v60,z0,tPen\WObj:=wPaper;
    MoveL Offs(pOrigin,115.64,105.98,0.00),v40,z0,tPen\WObj:=wPaper;
    MoveL Offs(pOrigin,114.58,105.98,0.00),v40,z0,tPen\WObj:=wPaper;
    MoveL Offs(pOrigin,114.58,95.02,0.00),v40,z0,tPen\WObj:=wPaper;
    MoveL Offs(pOrigin,113.53,94.87,0.00),v40,z0,tPen\WObj:=wPaper;
    MoveL Offs(pOrigin,113.53,105.82,0.00),v40,fine,tPen\WObj:=wPaper;
    MoveL Offs(pOrigin,113.53,105.82,6.00),v60,z5,tPen\WObj:=wPaper;
    MoveL Offs(pOrigin,112.47,104.78,6.00),vTravel,z5,tPen\WObj:=wPaper;
    MoveL Offs(pOrigin,112.47,104.78,0.00),v60,z0,tPen\WObj:=wPaper;
    MoveL Offs(pOrigin,112.47,94.87,0.00),v40,z0,tPen\WObj:=wPaper;
    MoveL Offs(pOrigin,111.42,94.87,0.00),v40,z0,tPen\WObj:=wPaper;
    MoveL Offs(pOrigin,111.42,103.72,0.00),v40,fine,tPen\WObj:=wPaper;
    MoveL Offs(pOrigin,111.42,103.72,6.00),v60,z5,tPen\WObj:=wPaper;
    MoveL Offs(pOrigin,110.36,102.82,6.00),vTravel,z5,tPen\WObj:=wPaper;
    MoveL Offs(pOrigin,110.36,102.82,0.00),v60,z0,tPen\WObj:=wPaper;
    MoveL Offs(pOrigin,110.36,94.87,0.00),v40,z0,tPen\WObj:=wPaper;
    MoveL Offs(pOrigin,109.30,95.32,0.00),v40,z0,tPen\WObj:=wPaper;
    MoveL Offs(pOrigin,109.30,102.38,0.00),v40,fine,tPen\WObj:=wPaper;
    MoveL Offs(pOrigin,109.30,102.38,6.00),v60,z5,tPen\WObj:=wPaper;
    MoveL Offs(pOrigin,107.75,103.35,6.00),vTravel,z5,tPen\WObj:=wPaper;
    MoveL Offs(pOrigin,107.75,103.35,0.00),v60,z0,tPen\WObj:=wPaper;
    MoveL Offs(pOrigin,131.30,103.35,0.00),v40,z0,tPen\WObj:=wPaper;
    MoveL Offs(pOrigin,132.04,103.33,0.00),v40,z0,tPen\WObj:=wPaper;
    MoveL Offs(pOrigin,121.64,92.93,0.00),v40,fine,tPen\WObj:=wPaper;
    MoveL Offs(pOrigin,121.64,92.93,6.00),v60,z5,tPen\WObj:=wPaper;
    MoveL Offs(pOrigin,120.15,92.94,6.00),vTravel,z5,tPen\WObj:=wPaper;
    MoveL Offs(pOrigin,120.15,92.94,0.00),v60,z0,tPen\WObj:=wPaper;
    MoveL Offs(pOrigin,132.03,104.82,0.00),v40,z0,tPen\WObj:=wPaper;
    MoveL Offs(pOrigin,132.54,104.54,0.00),v40,z0,tPen\WObj:=wPaper;
    MoveL Offs(pOrigin,106.03,131.06,0.00),v40,z0,tPen\WObj:=wPaper;
    MoveL Offs(pOrigin,106.96,130.52,0.00),v40,z0,tPen\WObj:=wPaper;
    MoveL Offs(pOrigin,109.72,133.28,0.00),v40,z0,tPen\WObj:=wPaper;
    MoveL Offs(pOrigin,108.91,134.15,0.00),v40,z0,tPen\WObj:=wPaper;
    MoveL Offs(pOrigin,132.56,110.50,0.00),v40,z0,tPen\WObj:=wPaper;
    MoveL Offs(pOrigin,131.81,110.56,0.00),v40,z0,tPen\WObj:=wPaper;
    MoveL Offs(pOrigin,114.20,92.95,0.00),v40,fine,tPen\WObj:=wPaper;
    MoveL Offs(pOrigin,114.20,92.95,6.00),v60,z5,tPen\WObj:=wPaper;
    MoveL Offs(pOrigin,113.04,91.19,6.00),vTravel,z5,tPen\WObj:=wPaper;
    MoveL Offs(pOrigin,113.04,91.19,0.00),v60,z0,tPen\WObj:=wPaper;
    MoveL Offs(pOrigin,132.56,71.68,0.00),v40,z0,tPen\WObj:=wPaper;
    MoveL Offs(pOrigin,131.81,71.74,0.00),v40,z0,tPen\WObj:=wPaper;
    MoveL Offs(pOrigin,110.81,50.73,0.00),v40,z0,tPen\WObj:=wPaper;
    MoveL Offs(pOrigin,111.22,49.70,0.00),v40,z0,tPen\WObj:=wPaper;
    MoveL Offs(pOrigin,106.13,54.79,0.00),v40,z0,tPen\WObj:=wPaper;
    MoveL Offs(pOrigin,106.97,54.36,0.00),v40,z0,tPen\WObj:=wPaper;
    MoveL Offs(pOrigin,131.89,79.29,0.00),v40,z0,tPen\WObj:=wPaper;
    MoveL Offs(pOrigin,132.58,79.12,0.00),v40,z0,tPen\WObj:=wPaper;
    MoveL Offs(pOrigin,120.59,91.11,0.00),v40,z0,tPen\WObj:=wPaper;
    MoveL Offs(pOrigin,120.80,90.59,0.00),v40,z0,tPen\WObj:=wPaper;
    MoveL Offs(pOrigin,107.12,76.91,0.00),v40,z0,tPen\WObj:=wPaper;
    MoveL Offs(pOrigin,108.05,76.95,0.00),v40,z0,tPen\WObj:=wPaper;
    MoveL Offs(pOrigin,131.00,76.95,0.00),v40,z0,tPen\WObj:=wPaper;
    MoveL Offs(pOrigin,131.00,75.90,0.00),v40,z0,tPen\WObj:=wPaper;
    MoveL Offs(pOrigin,108.05,75.90,0.00),v40,z0,tPen\WObj:=wPaper;
    MoveL Offs(pOrigin,107.90,74.84,0.00),v40,z0,tPen\WObj:=wPaper;
    MoveL Offs(pOrigin,131.00,74.84,0.00),v40,z0,tPen\WObj:=wPaper;
    MoveL Offs(pOrigin,131.80,74.71,0.00),v40,z0,tPen\WObj:=wPaper;
    MoveL Offs(pOrigin,107.94,50.85,0.00),v40,z0,tPen\WObj:=wPaper;
    MoveL Offs(pOrigin,108.20,51.61,0.00),v40,z0,tPen\WObj:=wPaper;
    MoveL Offs(pOrigin,131.00,51.61,0.00),v40,z0,tPen\WObj:=wPaper;
    MoveL Offs(pOrigin,131.45,52.66,0.00),v40,z0,tPen\WObj:=wPaper;
    MoveL Offs(pOrigin,107.75,52.66,0.00),v40,z0,tPen\WObj:=wPaper;
    MoveL Offs(pOrigin,106.87,52.77,0.00),v40,z0,tPen\WObj:=wPaper;
    MoveL Offs(pOrigin,131.79,77.69,0.00),v40,z0,tPen\WObj:=wPaper;
    MoveL Offs(pOrigin,132.47,77.74,0.00),v40,z0,tPen\WObj:=wPaper;
    MoveL Offs(pOrigin,119.10,91.10,0.00),v40,z0,tPen\WObj:=wPaper;
    MoveL Offs(pOrigin,119.20,90.49,0.00),v40,z0,tPen\WObj:=wPaper;
    MoveL Offs(pOrigin,107.11,78.40,0.00),v40,z0,tPen\WObj:=wPaper;
    MoveL Offs(pOrigin,108.05,78.01,0.00),v40,z0,tPen\WObj:=wPaper;
    MoveL Offs(pOrigin,131.00,78.01,0.00),v40,z0,tPen\WObj:=wPaper;
    MoveL Offs(pOrigin,131.00,79.06,0.00),v40,z0,tPen\WObj:=wPaper;
    MoveL Offs(pOrigin,108.05,79.06,0.00),v40,z0,tPen\WObj:=wPaper;
    MoveL Offs(pOrigin,108.05,80.12,0.00),v40,z0,tPen\WObj:=wPaper;
    MoveL Offs(pOrigin,131.15,80.12,0.00),v40,z0,tPen\WObj:=wPaper;
    MoveL Offs(pOrigin,131.15,81.18,0.00),v40,z0,tPen\WObj:=wPaper;
    MoveL Offs(pOrigin,108.05,81.18,0.00),v40,z0,tPen\WObj:=wPaper;
    MoveL Offs(pOrigin,108.05,82.23,0.00),v40,z0,tPen\WObj:=wPaper;
    MoveL Offs(pOrigin,131.00,82.23,0.00),v40,z0,tPen\WObj:=wPaper;
    MoveL Offs(pOrigin,131.15,83.29,0.00),v40,z0,tPen\WObj:=wPaper;
    MoveL Offs(pOrigin,108.05,83.29,0.00),v40,z0,tPen\WObj:=wPaper;
    MoveL Offs(pOrigin,107.10,82.87,0.00),v40,z0,tPen\WObj:=wPaper;
    MoveL Offs(pOrigin,114.84,90.61,0.00),v40,fine,tPen\WObj:=wPaper;
  ENDPROC

  PROC DrawPart17()
    MoveL Offs(pOrigin,114.84,90.61,6.00),v60,z5,tPen\WObj:=wPaper;
    MoveL Offs(pOrigin,116.33,90.61,6.00),vTravel,z5,tPen\WObj:=wPaper;
    MoveL Offs(pOrigin,116.33,90.61,0.00),v60,z0,tPen\WObj:=wPaper;
    MoveL Offs(pOrigin,106.89,81.17,0.00),v40,z0,tPen\WObj:=wPaper;
    MoveL Offs(pOrigin,106.10,81.71,0.00),v40,z0,tPen\WObj:=wPaper;
    MoveL Offs(pOrigin,132.83,54.98,0.00),v40,z0,tPen\WObj:=wPaper;
    MoveL Offs(pOrigin,132.07,55.57,0.00),v40,z0,tPen\WObj:=wPaper;
    MoveL Offs(pOrigin,127.19,50.69,0.00),v40,z0,tPen\WObj:=wPaper;
    MoveL Offs(pOrigin,127.60,49.75,0.00),v40,z0,tPen\WObj:=wPaper;
    MoveL Offs(pOrigin,106.07,71.28,0.00),v40,fine,tPen\WObj:=wPaper;
    MoveL Offs(pOrigin,106.07,71.28,6.00),v60,z5,tPen\WObj:=wPaper;
    MoveL Offs(pOrigin,106.92,72.23,6.00),vTravel,z5,tPen\WObj:=wPaper;
    MoveL Offs(pOrigin,106.92,72.23,0.00),v60,z0,tPen\WObj:=wPaper;
    MoveL Offs(pOrigin,125.16,90.48,0.00),v40,z0,tPen\WObj:=wPaper;
    MoveL Offs(pOrigin,125.27,90.91,0.00),v40,z0,tPen\WObj:=wPaper;
    MoveL Offs(pOrigin,132.48,83.70,0.00),v40,z0,tPen\WObj:=wPaper;
    MoveL Offs(pOrigin,131.88,83.75,0.00),v40,z0,tPen\WObj:=wPaper;
    MoveL Offs(pOrigin,106.96,58.83,0.00),v40,z0,tPen\WObj:=wPaper;
    MoveL Offs(pOrigin,107.90,59.00,0.00),v40,z0,tPen\WObj:=wPaper;
    MoveL Offs(pOrigin,131.15,59.00,0.00),v40,z0,tPen\WObj:=wPaper;
    MoveL Offs(pOrigin,132.06,58.55,0.00),v40,z0,tPen\WObj:=wPaper;
    MoveL Offs(pOrigin,124.21,50.70,0.00),v40,z0,tPen\WObj:=wPaper;
    MoveL Offs(pOrigin,124.62,49.74,0.00),v40,z0,tPen\WObj:=wPaper;
    MoveL Offs(pOrigin,106.17,68.20,0.00),v40,z0,tPen\WObj:=wPaper;
    MoveL Offs(pOrigin,106.93,67.76,0.00),v40,z0,tPen\WObj:=wPaper;
    MoveL Offs(pOrigin,129.63,90.46,0.00),v40,fine,tPen\WObj:=wPaper;
    MoveL Offs(pOrigin,129.63,90.46,6.00),v60,z5,tPen\WObj:=wPaper;
    MoveL Offs(pOrigin,128.04,91.13,6.00),vTravel,z5,tPen\WObj:=wPaper;
    MoveL Offs(pOrigin,128.04,91.13,0.00),v60,z0,tPen\WObj:=wPaper;
    MoveL Offs(pOrigin,132.81,86.36,0.00),v40,fine,tPen\WObj:=wPaper;
    MoveL Offs(pOrigin,132.81,86.36,6.00),v60,z5,tPen\WObj:=wPaper;
    MoveL Offs(pOrigin,131.15,86.46,6.00),vTravel,z5,tPen\WObj:=wPaper;
    MoveL Offs(pOrigin,131.15,86.46,0.00),v60,z0,tPen\WObj:=wPaper;
    MoveL Offs(pOrigin,107.90,86.46,0.00),v40,z0,tPen\WObj:=wPaper;
    MoveL Offs(pOrigin,107.90,85.40,0.00),v40,z0,tPen\WObj:=wPaper;
    MoveL Offs(pOrigin,131.15,85.40,0.00),v40,z0,tPen\WObj:=wPaper;
    MoveL Offs(pOrigin,131.15,84.34,0.00),v40,z0,tPen\WObj:=wPaper;
    MoveL Offs(pOrigin,108.05,84.34,0.00),v40,z0,tPen\WObj:=wPaper;
    MoveL Offs(pOrigin,107.10,84.36,0.00),v40,z0,tPen\WObj:=wPaper;
    MoveL Offs(pOrigin,113.35,90.62,0.00),v40,fine,tPen\WObj:=wPaper;
    MoveL Offs(pOrigin,113.35,90.62,6.00),v60,z5,tPen\WObj:=wPaper;
    MoveL Offs(pOrigin,111.76,90.51,6.00),vTravel,z5,tPen\WObj:=wPaper;
    MoveL Offs(pOrigin,111.76,90.51,0.00),v60,z0,tPen\WObj:=wPaper;
    MoveL Offs(pOrigin,106.88,85.63,0.00),v40,fine,tPen\WObj:=wPaper;
    MoveL Offs(pOrigin,106.88,85.63,6.00),v60,z5,tPen\WObj:=wPaper;
    MoveL Offs(pOrigin,105.90,86.39,6.00),vTravel,z5,tPen\WObj:=wPaper;
    MoveL Offs(pOrigin,105.90,86.39,0.00),v60,z0,tPen\WObj:=wPaper;
    MoveL Offs(pOrigin,132.95,59.34,0.00),v40,z0,tPen\WObj:=wPaper;
    MoveL Offs(pOrigin,132.06,60.03,0.00),v40,z0,tPen\WObj:=wPaper;
    MoveL Offs(pOrigin,122.72,50.70,0.00),v40,fine,tPen\WObj:=wPaper;
    MoveL Offs(pOrigin,122.72,50.70,6.00),v60,z5,tPen\WObj:=wPaper;
    MoveL Offs(pOrigin,123.35,49.53,6.00),vTravel,z5,tPen\WObj:=wPaper;
    MoveL Offs(pOrigin,123.35,49.53,0.00),v60,z0,tPen\WObj:=wPaper;
    MoveL Offs(pOrigin,105.84,67.03,0.00),v40,fine,tPen\WObj:=wPaper;
    MoveL Offs(pOrigin,105.84,67.03,6.00),v60,z5,tPen\WObj:=wPaper;
    MoveL Offs(pOrigin,107.90,67.45,6.00),vTravel,z5,tPen\WObj:=wPaper;
    MoveL Offs(pOrigin,107.90,67.45,0.00),v60,z0,tPen\WObj:=wPaper;
    MoveL Offs(pOrigin,131.15,67.45,0.00),v40,z0,tPen\WObj:=wPaper;
    MoveL Offs(pOrigin,131.82,67.27,0.00),v40,z0,tPen\WObj:=wPaper;
    MoveL Offs(pOrigin,115.28,50.72,0.00),v40,fine,tPen\WObj:=wPaper;
    MoveL Offs(pOrigin,115.28,50.72,6.00),v60,z5,tPen\WObj:=wPaper;
    MoveL Offs(pOrigin,115.90,49.50,6.00),vTravel,z5,tPen\WObj:=wPaper;
    MoveL Offs(pOrigin,115.90,49.50,0.00),v60,z0,tPen\WObj:=wPaper;
    MoveL Offs(pOrigin,105.72,59.69,0.00),v40,fine,tPen\WObj:=wPaper;
    MoveL Offs(pOrigin,105.72,59.69,6.00),v60,z5,tPen\WObj:=wPaper;
    MoveL Offs(pOrigin,106.04,60.86,6.00),vTravel,z5,tPen\WObj:=wPaper;
    MoveL Offs(pOrigin,106.04,60.86,0.00),v60,z0,tPen\WObj:=wPaper;
    MoveL Offs(pOrigin,117.28,49.61,0.00),v40,fine,tPen\WObj:=wPaper;
    MoveL Offs(pOrigin,117.28,49.61,6.00),v60,z5,tPen\WObj:=wPaper;
    MoveL Offs(pOrigin,116.77,50.72,6.00),vTravel,z5,tPen\WObj:=wPaper;
    MoveL Offs(pOrigin,116.77,50.72,0.00),v60,z0,tPen\WObj:=wPaper;
    MoveL Offs(pOrigin,132.04,65.99,0.00),v40,z0,tPen\WObj:=wPaper;
    MoveL Offs(pOrigin,132.75,65.51,0.00),v40,z0,tPen\WObj:=wPaper;
    MoveL Offs(pOrigin,107.08,91.18,0.00),v40,z0,tPen\WObj:=wPaper;
    MoveL Offs(pOrigin,106.44,90.32,0.00),v40,z0,tPen\WObj:=wPaper;
    MoveL Offs(pOrigin,132.53,64.23,0.00),v40,fine,tPen\WObj:=wPaper;
    MoveL Offs(pOrigin,132.53,64.23,6.00),v60,z5,tPen\WObj:=wPaper;
    MoveL Offs(pOrigin,134.02,64.23,6.00),vTravel,z5,tPen\WObj:=wPaper;
    MoveL Offs(pOrigin,134.02,64.23,0.00),v60,z0,tPen\WObj:=wPaper;
    MoveL Offs(pOrigin,147.28,50.98,0.00),v40,z0,tPen\WObj:=wPaper;
    MoveL Offs(pOrigin,148.35,51.40,0.00),v40,z0,tPen\WObj:=wPaper;
    MoveL Offs(pOrigin,133.92,65.83,0.00),v40,z0,tPen\WObj:=wPaper;
    MoveL Offs(pOrigin,134.80,65.77,0.00),v40,z0,tPen\WObj:=wPaper;
    MoveL Offs(pOrigin,159.62,90.59,0.00),v40,fine,tPen\WObj:=wPaper;
    MoveL Offs(pOrigin,159.62,90.59,6.00),v60,z5,tPen\WObj:=wPaper;
    MoveL Offs(pOrigin,161.01,90.48,6.00),vTravel,z5,tPen\WObj:=wPaper;
    MoveL Offs(pOrigin,161.01,90.48,0.00),v60,z0,tPen\WObj:=wPaper;
    MoveL Offs(pOrigin,134.81,64.28,0.00),v40,z0,tPen\WObj:=wPaper;
    MoveL Offs(pOrigin,135.80,64.28,0.00),v40,z0,tPen\WObj:=wPaper;
    MoveL Offs(pOrigin,160.85,64.28,0.00),v40,z0,tPen\WObj:=wPaper;
    MoveL Offs(pOrigin,161.72,64.31,0.00),v40,z0,tPen\WObj:=wPaper;
    MoveL Offs(pOrigin,151.22,53.81,0.00),v40,z0,tPen\WObj:=wPaper;
    MoveL Offs(pOrigin,151.33,52.90,0.00),v40,z0,tPen\WObj:=wPaper;
    MoveL Offs(pOrigin,134.15,70.09,0.00),v40,z0,tPen\WObj:=wPaper;
    MoveL Offs(pOrigin,134.79,70.24,0.00),v40,z0,tPen\WObj:=wPaper;
    MoveL Offs(pOrigin,155.05,90.50,0.00),v40,z0,tPen\WObj:=wPaper;
    MoveL Offs(pOrigin,155.16,90.89,0.00),v40,z0,tPen\WObj:=wPaper;
    MoveL Offs(pOrigin,165.56,80.49,0.00),v40,z0,tPen\WObj:=wPaper;
    MoveL Offs(pOrigin,164.76,80.79,0.00),v40,z0,tPen\WObj:=wPaper;
    MoveL Offs(pOrigin,135.06,51.09,0.00),v40,z0,tPen\WObj:=wPaper;
    MoveL Offs(pOrigin,135.80,51.61,0.00),v40,z0,tPen\WObj:=wPaper;
    MoveL Offs(pOrigin,142.25,51.61,0.00),v40,z0,tPen\WObj:=wPaper;
    MoveL Offs(pOrigin,142.40,50.96,0.00),v40,z0,tPen\WObj:=wPaper;
    MoveL Offs(pOrigin,164.57,73.13,0.00),v40,z0,tPen\WObj:=wPaper;
    MoveL Offs(pOrigin,165.43,73.15,0.00),v40,z0,tPen\WObj:=wPaper;
    MoveL Offs(pOrigin,147.72,90.87,0.00),v40,z0,tPen\WObj:=wPaper;
    MoveL Offs(pOrigin,147.39,90.31,0.00),v40,z0,tPen\WObj:=wPaper;
    MoveL Offs(pOrigin,134.77,77.68,0.00),v40,z0,tPen\WObj:=wPaper;
    MoveL Offs(pOrigin,134.17,77.53,0.00),v40,z0,tPen\WObj:=wPaper;
    MoveL Offs(pOrigin,155.81,55.89,0.00),v40,z0,tPen\WObj:=wPaper;
    MoveL Offs(pOrigin,156.66,56.53,0.00),v40,z0,tPen\WObj:=wPaper;
    MoveL Offs(pOrigin,134.07,79.13,0.00),v40,z0,tPen\WObj:=wPaper;
    MoveL Offs(pOrigin,134.77,79.17,0.00),v40,z0,tPen\WObj:=wPaper;
    MoveL Offs(pOrigin,145.90,90.31,0.00),v40,z0,tPen\WObj:=wPaper;
    MoveL Offs(pOrigin,146.23,90.86,0.00),v40,z0,tPen\WObj:=wPaper;
    MoveL Offs(pOrigin,165.11,71.98,0.00),v40,z0,tPen\WObj:=wPaper;
    MoveL Offs(pOrigin,164.25,71.32,0.00),v40,z0,tPen\WObj:=wPaper;
    MoveL Offs(pOrigin,144.21,51.28,0.00),v40,fine,tPen\WObj:=wPaper;
    MoveL Offs(pOrigin,144.21,51.28,6.00),v60,z5,tPen\WObj:=wPaper;
    MoveL Offs(pOrigin,146.12,51.70,6.00),vTravel,z5,tPen\WObj:=wPaper;
  ENDPROC

  PROC DrawPart18()
    MoveL Offs(pOrigin,146.12,51.70,0.00),v60,z0,tPen\WObj:=wPaper;
    MoveL Offs(pOrigin,163.73,69.30,0.00),v40,z0,tPen\WObj:=wPaper;
    MoveL Offs(pOrigin,163.10,69.56,0.00),v40,z0,tPen\WObj:=wPaper;
    MoveL Offs(pOrigin,135.80,69.56,0.00),v40,z0,tPen\WObj:=wPaper;
    MoveL Offs(pOrigin,135.80,70.62,0.00),v40,z0,tPen\WObj:=wPaper;
    MoveL Offs(pOrigin,163.40,70.62,0.00),v40,z0,tPen\WObj:=wPaper;
    MoveL Offs(pOrigin,163.55,71.67,0.00),v40,z0,tPen\WObj:=wPaper;
    MoveL Offs(pOrigin,135.80,71.67,0.00),v40,z0,tPen\WObj:=wPaper;
    MoveL Offs(pOrigin,134.79,71.73,0.00),v40,z0,tPen\WObj:=wPaper;
    MoveL Offs(pOrigin,153.56,90.50,0.00),v40,z0,tPen\WObj:=wPaper;
    MoveL Offs(pOrigin,153.67,90.88,0.00),v40,z0,tPen\WObj:=wPaper;
    MoveL Offs(pOrigin,165.76,78.79,0.00),v40,z0,tPen\WObj:=wPaper;
    MoveL Offs(pOrigin,165.08,78.13,0.00),v40,z0,tPen\WObj:=wPaper;
    MoveL Offs(pOrigin,137.61,50.66,0.00),v40,z0,tPen\WObj:=wPaper;
    MoveL Offs(pOrigin,138.13,49.67,0.00),v40,z0,tPen\WObj:=wPaper;
    MoveL Offs(pOrigin,133.78,54.02,0.00),v40,z0,tPen\WObj:=wPaper;
    MoveL Offs(pOrigin,134.52,53.54,0.00),v40,z0,tPen\WObj:=wPaper;
    MoveL Offs(pOrigin,164.43,83.45,0.00),v40,z0,tPen\WObj:=wPaper;
    MoveL Offs(pOrigin,163.70,83.29,0.00),v40,z0,tPen\WObj:=wPaper;
    MoveL Offs(pOrigin,135.80,83.29,0.00),v40,z0,tPen\WObj:=wPaper;
    MoveL Offs(pOrigin,134.86,83.75,0.00),v40,z0,tPen\WObj:=wPaper;
    MoveL Offs(pOrigin,141.33,90.22,0.00),v40,z0,tPen\WObj:=wPaper;
    MoveL Offs(pOrigin,141.76,90.85,0.00),v40,z0,tPen\WObj:=wPaper;
    MoveL Offs(pOrigin,164.46,68.15,0.00),v40,z0,tPen\WObj:=wPaper;
    MoveL Offs(pOrigin,163.82,67.30,0.00),v40,z0,tPen\WObj:=wPaper;
    MoveL Offs(pOrigin,140.27,90.84,0.00),v40,z0,tPen\WObj:=wPaper;
    MoveL Offs(pOrigin,139.84,90.22,0.00),v40,z0,tPen\WObj:=wPaper;
    MoveL Offs(pOrigin,134.86,85.24,0.00),v40,z0,tPen\WObj:=wPaper;
    MoveL Offs(pOrigin,134.19,84.98,0.00),v40,z0,tPen\WObj:=wPaper;
    MoveL Offs(pOrigin,159.65,59.52,0.00),v40,z0,tPen\WObj:=wPaper;
    MoveL Offs(pOrigin,158.90,60.08,0.00),v40,z0,tPen\WObj:=wPaper;
    MoveL Offs(pOrigin,159.35,60.53,0.00),v40,z0,tPen\WObj:=wPaper;
    MoveL Offs(pOrigin,158.90,60.08,0.00),v40,z0,tPen\WObj:=wPaper;
    MoveL Offs(pOrigin,158.60,61.11,0.00),v40,z0,tPen\WObj:=wPaper;
    MoveL Offs(pOrigin,135.65,61.11,0.00),v40,z0,tPen\WObj:=wPaper;
    MoveL Offs(pOrigin,135.65,62.17,0.00),v40,z0,tPen\WObj:=wPaper;
    MoveL Offs(pOrigin,159.50,62.17,0.00),v40,fine,tPen\WObj:=wPaper;
    MoveL Offs(pOrigin,159.50,62.17,6.00),v60,z5,tPen\WObj:=wPaper;
    MoveL Offs(pOrigin,160.10,63.22,6.00),vTravel,z5,tPen\WObj:=wPaper;
    MoveL Offs(pOrigin,160.10,63.22,0.00),v60,z0,tPen\WObj:=wPaper;
    MoveL Offs(pOrigin,135.65,63.22,0.00),v40,z0,tPen\WObj:=wPaper;
    MoveL Offs(pOrigin,134.81,62.79,0.00),v40,z0,tPen\WObj:=wPaper;
    MoveL Offs(pOrigin,161.86,89.84,0.00),v40,z0,tPen\WObj:=wPaper;
    MoveL Offs(pOrigin,160.70,89.62,0.00),v40,z0,tPen\WObj:=wPaper;
    MoveL Offs(pOrigin,148.55,89.62,0.00),v40,z0,tPen\WObj:=wPaper;
    MoveL Offs(pOrigin,149.09,90.51,0.00),v40,z0,tPen\WObj:=wPaper;
    MoveL Offs(pOrigin,134.78,76.19,0.00),v40,z0,tPen\WObj:=wPaper;
    MoveL Offs(pOrigin,134.16,76.04,0.00),v40,z0,tPen\WObj:=wPaper;
    MoveL Offs(pOrigin,154.85,55.36,0.00),v40,z0,tPen\WObj:=wPaper;
    MoveL Offs(pOrigin,154.10,55.58,0.00),v40,z0,tPen\WObj:=wPaper;
    MoveL Offs(pOrigin,154.85,56.17,0.00),v40,z0,tPen\WObj:=wPaper;
    MoveL Offs(pOrigin,154.10,55.58,0.00),v40,z0,tPen\WObj:=wPaper;
    MoveL Offs(pOrigin,154.10,54.61,0.00),v40,z0,tPen\WObj:=wPaper;
    MoveL Offs(pOrigin,134.05,74.66,0.00),v40,fine,tPen\WObj:=wPaper;
    MoveL Offs(pOrigin,134.05,74.66,6.00),v60,z5,tPen\WObj:=wPaper;
    MoveL Offs(pOrigin,133.94,73.28,6.00),vTravel,z5,tPen\WObj:=wPaper;
    MoveL Offs(pOrigin,133.94,73.28,0.00),v60,z0,tPen\WObj:=wPaper;
    MoveL Offs(pOrigin,153.25,53.97,0.00),v40,z0,tPen\WObj:=wPaper;
    MoveL Offs(pOrigin,152.29,53.44,0.00),v40,z0,tPen\WObj:=wPaper;
    MoveL Offs(pOrigin,134.05,71.68,0.00),v40,fine,tPen\WObj:=wPaper;
    MoveL Offs(pOrigin,134.05,71.68,6.00),v60,z5,tPen\WObj:=wPaper;
    MoveL Offs(pOrigin,134.78,73.22,6.00),vTravel,z5,tPen\WObj:=wPaper;
    MoveL Offs(pOrigin,134.78,73.22,0.00),v60,z0,tPen\WObj:=wPaper;
    MoveL Offs(pOrigin,152.07,90.50,0.00),v40,z0,tPen\WObj:=wPaper;
    MoveL Offs(pOrigin,151.97,91.09,0.00),v40,z0,tPen\WObj:=wPaper;
    MoveL Offs(pOrigin,165.87,77.20,0.00),v40,fine,tPen\WObj:=wPaper;
    MoveL Offs(pOrigin,165.87,77.20,6.00),v60,z5,tPen\WObj:=wPaper;
    MoveL Offs(pOrigin,164.15,76.95,6.00),vTravel,z5,tPen\WObj:=wPaper;
    MoveL Offs(pOrigin,164.15,76.95,0.00),v60,z0,tPen\WObj:=wPaper;
    MoveL Offs(pOrigin,135.80,76.95,0.00),v40,z0,tPen\WObj:=wPaper;
    MoveL Offs(pOrigin,135.80,75.90,0.00),v40,z0,tPen\WObj:=wPaper;
    MoveL Offs(pOrigin,164.15,75.90,0.00),v40,fine,tPen\WObj:=wPaper;
    MoveL Offs(pOrigin,164.15,75.90,6.00),v60,z5,tPen\WObj:=wPaper;
    MoveL Offs(pOrigin,165.54,74.54,6.00),vTravel,z5,tPen\WObj:=wPaper;
    MoveL Offs(pOrigin,165.54,74.54,0.00),v60,z0,tPen\WObj:=wPaper;
    MoveL Offs(pOrigin,149.20,90.87,0.00),v40,fine,tPen\WObj:=wPaper;
    MoveL Offs(pOrigin,149.20,90.87,6.00),v60,z5,tPen\WObj:=wPaper;
    MoveL Offs(pOrigin,149.31,92.25,6.00),vTravel,z5,tPen\WObj:=wPaper;
    MoveL Offs(pOrigin,149.31,92.25,0.00),v60,z0,tPen\WObj:=wPaper;
    MoveL Offs(pOrigin,133.94,107.63,0.00),v40,z0,tPen\WObj:=wPaper;
    MoveL Offs(pOrigin,134.69,107.47,0.00),v40,z0,tPen\WObj:=wPaper;
    MoveL Offs(pOrigin,153.88,126.66,0.00),v40,z0,tPen\WObj:=wPaper;
    MoveL Offs(pOrigin,153.14,127.41,0.00),v40,z0,tPen\WObj:=wPaper;
    MoveL Offs(pOrigin,134.68,108.96,0.00),v40,z0,tPen\WObj:=wPaper;
    MoveL Offs(pOrigin,133.94,109.12,0.00),v40,z0,tPen\WObj:=wPaper;
    MoveL Offs(pOrigin,151.02,92.04,0.00),v40,z0,tPen\WObj:=wPaper;
    MoveL Offs(pOrigin,151.53,92.95,0.00),v40,z0,tPen\WObj:=wPaper;
    MoveL Offs(pOrigin,155.99,97.41,0.00),v40,z0,tPen\WObj:=wPaper;
    MoveL Offs(pOrigin,156.73,96.66,0.00),v40,z0,tPen\WObj:=wPaper;
    MoveL Offs(pOrigin,153.23,93.16,0.00),v40,z0,tPen\WObj:=wPaper;
    MoveL Offs(pOrigin,153.78,92.27,0.00),v40,z0,tPen\WObj:=wPaper;
    MoveL Offs(pOrigin,134.16,111.89,0.00),v40,z0,tPen\WObj:=wPaper;
    MoveL Offs(pOrigin,134.78,112.04,0.00),v40,z0,tPen\WObj:=wPaper;
    MoveL Offs(pOrigin,151.64,128.91,0.00),v40,z0,tPen\WObj:=wPaper;
    MoveL Offs(pOrigin,152.50,128.26,0.00),v40,z0,tPen\WObj:=wPaper;
    MoveL Offs(pOrigin,134.78,110.55,0.00),v40,z0,tPen\WObj:=wPaper;
    MoveL Offs(pOrigin,134.60,110.47,0.00),v40,z0,tPen\WObj:=wPaper;
    MoveL Offs(pOrigin,134.60,130.12,0.00),v40,z0,tPen\WObj:=wPaper;
    MoveL Offs(pOrigin,134.60,110.47,0.00),v40,z0,tPen\WObj:=wPaper;
    MoveL Offs(pOrigin,134.05,110.50,0.00),v40,z0,tPen\WObj:=wPaper;
    MoveL Offs(pOrigin,152.29,92.26,0.00),v40,fine,tPen\WObj:=wPaper;
    MoveL Offs(pOrigin,152.29,92.26,6.00),v60,z5,tPen\WObj:=wPaper;
    MoveL Offs(pOrigin,150.04,92.96,6.00),vTravel,z5,tPen\WObj:=wPaper;
    MoveL Offs(pOrigin,150.04,92.96,0.00),v60,z0,tPen\WObj:=wPaper;
    MoveL Offs(pOrigin,155.03,97.94,0.00),v40,z0,tPen\WObj:=wPaper;
    MoveL Offs(pOrigin,155.00,97.02,0.00),v40,z0,tPen\WObj:=wPaper;
    MoveL Offs(pOrigin,135.35,97.02,0.00),v40,z0,tPen\WObj:=wPaper;
    MoveL Offs(pOrigin,135.35,95.96,0.00),v40,z0,tPen\WObj:=wPaper;
    MoveL Offs(pOrigin,156.20,95.96,0.00),v40,fine,tPen\WObj:=wPaper;
    MoveL Offs(pOrigin,156.20,95.96,6.00),v60,z5,tPen\WObj:=wPaper;
    MoveL Offs(pOrigin,157.48,95.91,6.00),vTravel,z5,tPen\WObj:=wPaper;
    MoveL Offs(pOrigin,157.48,95.91,0.00),v60,z0,tPen\WObj:=wPaper;
    MoveL Offs(pOrigin,154.72,93.16,0.00),v40,fine,tPen\WObj:=wPaper;
    MoveL Offs(pOrigin,154.72,93.16,6.00),v60,z5,tPen\WObj:=wPaper;
    MoveL Offs(pOrigin,153.66,94.87,6.00),vTravel,z5,tPen\WObj:=wPaper;
    MoveL Offs(pOrigin,153.66,94.87,0.00),v60,z0,tPen\WObj:=wPaper;
    MoveL Offs(pOrigin,153.66,96.82,0.00),v40,fine,tPen\WObj:=wPaper;
    MoveL Offs(pOrigin,153.66,96.82,6.00),v60,z5,tPen\WObj:=wPaper;
    MoveL Offs(pOrigin,153.65,98.07,6.00),vTravel,z5,tPen\WObj:=wPaper;
    MoveL Offs(pOrigin,153.65,98.07,0.00),v60,z0,tPen\WObj:=wPaper;
  ENDPROC

  PROC DrawPart19()
    MoveL Offs(pOrigin,135.35,98.07,0.00),v40,z0,tPen\WObj:=wPaper;
    MoveL Offs(pOrigin,135.35,99.13,0.00),v40,z0,tPen\WObj:=wPaper;
    MoveL Offs(pOrigin,152.15,99.13,0.00),v40,z0,tPen\WObj:=wPaper;
    MoveL Offs(pOrigin,152.47,99.86,0.00),v40,z0,tPen\WObj:=wPaper;
    MoveL Offs(pOrigin,145.68,93.08,0.00),v40,z0,tPen\WObj:=wPaper;
    MoveL Offs(pOrigin,146.23,92.35,0.00),v40,z0,tPen\WObj:=wPaper;
    MoveL Offs(pOrigin,134.14,104.44,0.00),v40,z0,tPen\WObj:=wPaper;
    MoveL Offs(pOrigin,134.80,104.59,0.00),v40,z0,tPen\WObj:=wPaper;
    MoveL Offs(pOrigin,155.06,124.85,0.00),v40,z0,tPen\WObj:=wPaper;
    MoveL Offs(pOrigin,154.25,124.47,0.00),v40,z0,tPen\WObj:=wPaper;
    MoveL Offs(pOrigin,135.65,124.47,0.00),v40,z0,tPen\WObj:=wPaper;
    MoveL Offs(pOrigin,134.75,123.95,0.00),v40,z0,tPen\WObj:=wPaper;
    MoveL Offs(pOrigin,143.76,132.97,0.00),v40,z0,tPen\WObj:=wPaper;
    MoveL Offs(pOrigin,143.48,133.93,0.00),v40,z0,tPen\WObj:=wPaper;
    MoveL Offs(pOrigin,158.22,119.19,0.00),v40,fine,tPen\WObj:=wPaper;
    MoveL Offs(pOrigin,158.22,119.19,6.00),v60,z5,tPen\WObj:=wPaper;
    MoveL Offs(pOrigin,156.50,119.19,6.00),vTravel,z5,tPen\WObj:=wPaper;
    MoveL Offs(pOrigin,156.50,119.19,0.00),v60,z0,tPen\WObj:=wPaper;
    MoveL Offs(pOrigin,135.65,119.19,0.00),v40,z0,tPen\WObj:=wPaper;
    MoveL Offs(pOrigin,135.65,118.14,0.00),v40,z0,tPen\WObj:=wPaper;
    MoveL Offs(pOrigin,156.65,118.14,0.00),v40,z0,tPen\WObj:=wPaper;
    MoveL Offs(pOrigin,156.80,117.08,0.00),v40,z0,tPen\WObj:=wPaper;
    MoveL Offs(pOrigin,135.65,117.08,0.00),v40,z0,tPen\WObj:=wPaper;
    MoveL Offs(pOrigin,135.65,116.02,0.00),v40,z0,tPen\WObj:=wPaper;
    MoveL Offs(pOrigin,156.80,116.02,0.00),v40,z0,tPen\WObj:=wPaper;
    MoveL Offs(pOrigin,156.65,114.97,0.00),v40,z0,tPen\WObj:=wPaper;
    MoveL Offs(pOrigin,135.65,114.97,0.00),v40,z0,tPen\WObj:=wPaper;
    MoveL Offs(pOrigin,134.77,115.02,0.00),v40,z0,tPen\WObj:=wPaper;
    MoveL Offs(pOrigin,150.04,130.29,0.00),v40,z0,tPen\WObj:=wPaper;
    MoveL Offs(pOrigin,149.30,129.75,0.00),v40,z0,tPen\WObj:=wPaper;
    MoveL Offs(pOrigin,135.35,129.75,0.00),v40,z0,tPen\WObj:=wPaper;
    MoveL Offs(pOrigin,134.41,129.59,0.00),v40,z0,tPen\WObj:=wPaper;
    MoveL Offs(pOrigin,138.12,133.30,0.00),v40,fine,tPen\WObj:=wPaper;
    MoveL Offs(pOrigin,138.12,133.30,6.00),v60,z5,tPen\WObj:=wPaper;
    MoveL Offs(pOrigin,137.82,131.47,6.00),vTravel,z5,tPen\WObj:=wPaper;
    MoveL Offs(pOrigin,137.82,131.47,0.00),v60,z0,tPen\WObj:=wPaper;
    MoveL Offs(pOrigin,137.82,128.92,0.00),v40,fine,tPen\WObj:=wPaper;
    MoveL Offs(pOrigin,137.82,128.92,6.00),v60,z5,tPen\WObj:=wPaper;
    MoveL Offs(pOrigin,136.76,128.32,6.00),vTravel,z5,tPen\WObj:=wPaper;
    MoveL Offs(pOrigin,136.76,128.32,0.00),v60,z0,tPen\WObj:=wPaper;
    MoveL Offs(pOrigin,136.76,131.47,0.00),v40,fine,tPen\WObj:=wPaper;
    MoveL Offs(pOrigin,136.76,131.47,6.00),v60,z5,tPen\WObj:=wPaper;
    MoveL Offs(pOrigin,135.50,131.86,6.00),vTravel,z5,tPen\WObj:=wPaper;
    MoveL Offs(pOrigin,135.50,131.86,0.00),v60,z0,tPen\WObj:=wPaper;
    MoveL Offs(pOrigin,144.65,131.86,0.00),v40,z0,tPen\WObj:=wPaper;
    MoveL Offs(pOrigin,144.93,132.65,0.00),v40,z0,tPen\WObj:=wPaper;
    MoveL Offs(pOrigin,134.75,122.46,0.00),v40,z0,tPen\WObj:=wPaper;
    MoveL Offs(pOrigin,135.65,122.36,0.00),v40,z0,tPen\WObj:=wPaper;
    MoveL Offs(pOrigin,155.45,122.36,0.00),v40,z0,tPen\WObj:=wPaper;
    MoveL Offs(pOrigin,156.02,122.83,0.00),v40,z0,tPen\WObj:=wPaper;
    MoveL Offs(pOrigin,134.49,101.30,0.00),v40,z0,tPen\WObj:=wPaper;
    MoveL Offs(pOrigin,133.92,101.68,0.00),v40,z0,tPen\WObj:=wPaper;
    MoveL Offs(pOrigin,143.36,92.24,0.00),v40,z0,tPen\WObj:=wPaper;
    MoveL Offs(pOrigin,142.70,93.08,0.00),v40,z0,tPen\WObj:=wPaper;
    MoveL Offs(pOrigin,150.98,101.36,0.00),v40,z0,tPen\WObj:=wPaper;
    MoveL Offs(pOrigin,150.50,101.32,0.00),v40,z0,tPen\WObj:=wPaper;
    MoveL Offs(pOrigin,151.10,100.68,0.00),v40,z0,tPen\WObj:=wPaper;
    MoveL Offs(pOrigin,151.80,102.57,0.00),v40,z0,tPen\WObj:=wPaper;
    MoveL Offs(pOrigin,150.50,101.32,0.00),v40,z0,tPen\WObj:=wPaper;
    MoveL Offs(pOrigin,150.05,101.24,0.00),v40,z0,tPen\WObj:=wPaper;
    MoveL Offs(pOrigin,135.35,101.24,0.00),v40,z0,tPen\WObj:=wPaper;
    MoveL Offs(pOrigin,135.35,102.30,0.00),v40,z0,tPen\WObj:=wPaper;
    MoveL Offs(pOrigin,150.50,102.30,0.00),v40,z0,tPen\WObj:=wPaper;
    MoveL Offs(pOrigin,149.43,102.68,0.00),v40,z0,tPen\WObj:=wPaper;
    MoveL Offs(pOrigin,149.43,104.02,0.00),v40,fine,tPen\WObj:=wPaper;
    MoveL Offs(pOrigin,149.43,104.02,6.00),v60,z5,tPen\WObj:=wPaper;
    MoveL Offs(pOrigin,148.38,102.68,6.00),vTravel,z5,tPen\WObj:=wPaper;
    MoveL Offs(pOrigin,148.38,102.68,0.00),v60,z0,tPen\WObj:=wPaper;
    MoveL Offs(pOrigin,148.38,94.72,0.00),v40,z0,tPen\WObj:=wPaper;
    MoveL Offs(pOrigin,149.43,94.72,0.00),v40,z0,tPen\WObj:=wPaper;
    MoveL Offs(pOrigin,149.43,99.98,0.00),v40,z0,tPen\WObj:=wPaper;
    MoveL Offs(pOrigin,150.50,100.18,0.00),v40,z0,tPen\WObj:=wPaper;
    MoveL Offs(pOrigin,135.35,100.18,0.00),v40,z0,tPen\WObj:=wPaper;
    MoveL Offs(pOrigin,134.71,100.02,0.00),v40,z0,tPen\WObj:=wPaper;
    MoveL Offs(pOrigin,156.45,121.76,0.00),v40,z0,tPen\WObj:=wPaper;
    MoveL Offs(pOrigin,155.90,121.30,0.00),v40,z0,tPen\WObj:=wPaper;
    MoveL Offs(pOrigin,135.65,121.30,0.00),v40,z0,tPen\WObj:=wPaper;
    MoveL Offs(pOrigin,134.75,120.98,0.00),v40,z0,tPen\WObj:=wPaper;
    MoveL Offs(pOrigin,146.00,132.22,0.00),v40,z0,tPen\WObj:=wPaper;
    MoveL Offs(pOrigin,145.81,133.09,0.00),v40,z0,tPen\WObj:=wPaper;
    MoveL Offs(pOrigin,157.38,121.53,0.00),v40,fine,tPen\WObj:=wPaper;
    MoveL Offs(pOrigin,157.38,121.53,6.00),v60,z5,tPen\WObj:=wPaper;
    MoveL Offs(pOrigin,156.43,123.97,6.00),vTravel,z5,tPen\WObj:=wPaper;
    MoveL Offs(pOrigin,156.43,123.97,0.00),v60,z0,tPen\WObj:=wPaper;
    MoveL Offs(pOrigin,148.36,132.03,0.00),v40,z0,tPen\WObj:=wPaper;
    MoveL Offs(pOrigin,148.13,131.36,0.00),v40,z0,tPen\WObj:=wPaper;
    MoveL Offs(pOrigin,134.76,118.00,0.00),v40,z0,tPen\WObj:=wPaper;
    MoveL Offs(pOrigin,134.07,117.95,0.00),v40,z0,tPen\WObj:=wPaper;
    MoveL Offs(pOrigin,159.63,92.39,0.00),v40,z0,tPen\WObj:=wPaper;
    MoveL Offs(pOrigin,160.38,93.14,0.00),v40,z0,tPen\WObj:=wPaper;
    MoveL Offs(pOrigin,153.70,99.82,0.00),v40,z0,tPen\WObj:=wPaper;
    MoveL Offs(pOrigin,153.32,99.22,0.00),v40,z0,tPen\WObj:=wPaper;
    MoveL Offs(pOrigin,147.28,93.18,0.00),v40,z0,tPen\WObj:=wPaper;
    MoveL Offs(pOrigin,147.72,92.35,0.00),v40,z0,tPen\WObj:=wPaper;
    MoveL Offs(pOrigin,134.04,106.04,0.00),v40,fine,tPen\WObj:=wPaper;
    MoveL Offs(pOrigin,134.04,106.04,6.00),v60,z5,tPen\WObj:=wPaper;
    MoveL Offs(pOrigin,135.65,106.52,6.00),vTravel,z5,tPen\WObj:=wPaper;
    MoveL Offs(pOrigin,135.65,106.52,0.00),v60,z0,tPen\WObj:=wPaper;
    MoveL Offs(pOrigin,154.25,106.52,0.00),v40,fine,tPen\WObj:=wPaper;
    MoveL Offs(pOrigin,154.25,106.52,6.00),v60,z5,tPen\WObj:=wPaper;
    MoveL Offs(pOrigin,155.00,107.58,6.00),vTravel,z5,tPen\WObj:=wPaper;
    MoveL Offs(pOrigin,155.00,107.58,0.00),v60,z0,tPen\WObj:=wPaper;
    MoveL Offs(pOrigin,135.50,107.58,0.00),v40,z0,tPen\WObj:=wPaper;
    MoveL Offs(pOrigin,135.50,108.63,0.00),v40,z0,tPen\WObj:=wPaper;
    MoveL Offs(pOrigin,155.45,108.63,0.00),v40,z0,tPen\WObj:=wPaper;
    MoveL Offs(pOrigin,156.35,108.53,0.00),v40,z0,tPen\WObj:=wPaper;
    MoveL Offs(pOrigin,157.20,110.78,0.00),v40,z0,tPen\WObj:=wPaper;
    MoveL Offs(pOrigin,156.35,108.53,0.00),v40,z0,tPen\WObj:=wPaper;
    MoveL Offs(pOrigin,156.81,108.65,0.00),v40,z0,tPen\WObj:=wPaper;
    MoveL Offs(pOrigin,133.68,131.78,0.00),v40,z0,tPen\WObj:=wPaper;
    MoveL Offs(pOrigin,134.11,132.84,0.00),v40,z0,tPen\WObj:=wPaper;
    MoveL Offs(pOrigin,157.45,109.51,0.00),v40,fine,tPen\WObj:=wPaper;
    MoveL Offs(pOrigin,157.45,109.51,6.00),v60,z5,tPen\WObj:=wPaper;
    MoveL Offs(pOrigin,155.90,109.69,6.00),vTravel,z5,tPen\WObj:=wPaper;
    MoveL Offs(pOrigin,155.90,109.69,0.00),v60,z0,tPen\WObj:=wPaper;
    MoveL Offs(pOrigin,135.65,109.69,0.00),v40,z0,tPen\WObj:=wPaper;
    MoveL Offs(pOrigin,135.65,110.74,0.00),v40,z0,tPen\WObj:=wPaper;
    MoveL Offs(pOrigin,156.20,110.74,0.00),v40,z0,tPen\WObj:=wPaper;
    MoveL Offs(pOrigin,156.50,111.80,0.00),v40,z0,tPen\WObj:=wPaper;
    MoveL Offs(pOrigin,135.65,111.80,0.00),v40,z0,tPen\WObj:=wPaper;
  ENDPROC

  PROC DrawPart20()
    MoveL Offs(pOrigin,135.80,112.86,0.00),v40,z0,tPen\WObj:=wPaper;
    MoveL Offs(pOrigin,156.65,112.86,0.00),v40,z0,tPen\WObj:=wPaper;
    MoveL Offs(pOrigin,156.65,113.91,0.00),v40,z0,tPen\WObj:=wPaper;
    MoveL Offs(pOrigin,135.80,113.91,0.00),v40,fine,tPen\WObj:=wPaper;
    MoveL Offs(pOrigin,135.80,113.91,6.00),v60,z5,tPen\WObj:=wPaper;
    MoveL Offs(pOrigin,133.96,115.08,6.00),vTravel,z5,tPen\WObj:=wPaper;
    MoveL Offs(pOrigin,133.96,115.08,0.00),v60,z0,tPen\WObj:=wPaper;
    MoveL Offs(pOrigin,165.46,83.58,0.00),v40,fine,tPen\WObj:=wPaper;
    MoveL Offs(pOrigin,165.46,83.58,6.00),v60,z5,tPen\WObj:=wPaper;
    MoveL Offs(pOrigin,164.75,82.28,6.00),vTravel,z5,tPen\WObj:=wPaper;
    MoveL Offs(pOrigin,164.75,82.28,0.00),v60,z0,tPen\WObj:=wPaper;
    MoveL Offs(pOrigin,134.52,52.05,0.00),v40,z0,tPen\WObj:=wPaper;
    MoveL Offs(pOrigin,135.35,52.66,0.00),v40,z0,tPen\WObj:=wPaper;
    MoveL Offs(pOrigin,146.90,52.66,0.00),v40,fine,tPen\WObj:=wPaper;
    MoveL Offs(pOrigin,146.90,52.66,6.00),v60,z5,tPen\WObj:=wPaper;
    MoveL Offs(pOrigin,146.11,50.65,6.00),vTravel,z5,tPen\WObj:=wPaper;
    MoveL Offs(pOrigin,146.11,50.65,0.00),v60,z0,tPen\WObj:=wPaper;
    MoveL Offs(pOrigin,134.13,62.64,0.00),v40,fine,tPen\WObj:=wPaper;
    MoveL Offs(pOrigin,134.13,62.64,6.00),v60,z5,tPen\WObj:=wPaper;
    MoveL Offs(pOrigin,135.65,60.06,6.00),vTravel,z5,tPen\WObj:=wPaper;
    MoveL Offs(pOrigin,135.65,60.06,0.00),v60,z0,tPen\WObj:=wPaper;
    MoveL Offs(pOrigin,157.70,60.06,0.00),v40,z0,tPen\WObj:=wPaper;
    MoveL Offs(pOrigin,157.80,58.90,0.00),v40,z0,tPen\WObj:=wPaper;
    MoveL Offs(pOrigin,156.00,57.09,0.00),v40,z0,tPen\WObj:=wPaper;
    MoveL Offs(pOrigin,155.90,57.08,0.00),v40,z0,tPen\WObj:=wPaper;
    MoveL Offs(pOrigin,156.95,57.97,0.00),v40,z0,tPen\WObj:=wPaper;
    MoveL Offs(pOrigin,155.90,57.08,0.00),v40,z0,tPen\WObj:=wPaper;
    MoveL Offs(pOrigin,155.75,57.94,0.00),v40,z0,tPen\WObj:=wPaper;
    MoveL Offs(pOrigin,135.50,57.94,0.00),v40,z0,tPen\WObj:=wPaper;
    MoveL Offs(pOrigin,134.72,58.22,0.00),v40,z0,tPen\WObj:=wPaper;
    MoveL Offs(pOrigin,163.36,86.86,0.00),v40,fine,tPen\WObj:=wPaper;
    MoveL Offs(pOrigin,163.36,86.86,6.00),v60,z5,tPen\WObj:=wPaper;
    MoveL Offs(pOrigin,163.56,88.46,6.00),vTravel,z5,tPen\WObj:=wPaper;
    MoveL Offs(pOrigin,163.56,88.46,0.00),v60,z0,tPen\WObj:=wPaper;
    MoveL Offs(pOrigin,161.12,90.90,0.00),v40,fine,tPen\WObj:=wPaper;
    MoveL Offs(pOrigin,161.12,90.90,6.00),v60,z5,tPen\WObj:=wPaper;
    MoveL Offs(pOrigin,158.57,91.96,6.00),vTravel,z5,tPen\WObj:=wPaper;
    MoveL Offs(pOrigin,158.57,91.96,0.00),v60,z0,tPen\WObj:=wPaper;
    MoveL Offs(pOrigin,134.07,116.46,0.00),v40,z0,tPen\WObj:=wPaper;
    MoveL Offs(pOrigin,134.66,116.40,0.00),v40,z0,tPen\WObj:=wPaper;
    MoveL Offs(pOrigin,149.09,130.83,0.00),v40,fine,tPen\WObj:=wPaper;
    MoveL Offs(pOrigin,149.09,130.83,6.00),v60,z5,tPen\WObj:=wPaper;
    MoveL Offs(pOrigin,148.38,128.93,6.00),vTravel,z5,tPen\WObj:=wPaper;
    MoveL Offs(pOrigin,148.38,128.93,0.00),v60,z0,tPen\WObj:=wPaper;
    MoveL Offs(pOrigin,148.38,127.42,0.00),v40,fine,tPen\WObj:=wPaper;
    MoveL Offs(pOrigin,148.38,127.42,6.00),v60,z5,tPen\WObj:=wPaper;
    MoveL Offs(pOrigin,147.32,126.52,6.00),vTravel,z5,tPen\WObj:=wPaper;
    MoveL Offs(pOrigin,147.32,126.52,0.00),v60,z0,tPen\WObj:=wPaper;
    MoveL Offs(pOrigin,147.32,129.52,0.00),v40,fine,tPen\WObj:=wPaper;
    MoveL Offs(pOrigin,147.32,129.52,6.00),v60,z5,tPen\WObj:=wPaper;
    MoveL Offs(pOrigin,146.26,130.12,6.00),vTravel,z5,tPen\WObj:=wPaper;
    MoveL Offs(pOrigin,146.26,130.12,0.00),v60,z0,tPen\WObj:=wPaper;
    MoveL Offs(pOrigin,146.26,126.08,0.00),v40,fine,tPen\WObj:=wPaper;
    MoveL Offs(pOrigin,146.26,126.08,6.00),v60,z5,tPen\WObj:=wPaper;
    MoveL Offs(pOrigin,145.21,124.58,6.00),vTravel,z5,tPen\WObj:=wPaper;
    MoveL Offs(pOrigin,145.21,124.58,0.00),v60,z0,tPen\WObj:=wPaper;
    MoveL Offs(pOrigin,145.21,130.57,0.00),v40,z0,tPen\WObj:=wPaper;
    MoveL Offs(pOrigin,144.15,130.57,0.00),v40,z0,tPen\WObj:=wPaper;
    MoveL Offs(pOrigin,144.15,124.42,0.00),v40,z0,tPen\WObj:=wPaper;
    MoveL Offs(pOrigin,143.10,124.42,0.00),v40,z0,tPen\WObj:=wPaper;
    MoveL Offs(pOrigin,143.10,129.22,0.00),v40,fine,tPen\WObj:=wPaper;
    MoveL Offs(pOrigin,143.10,129.22,6.00),v60,z5,tPen\WObj:=wPaper;
    MoveL Offs(pOrigin,142.04,127.88,6.00),vTravel,z5,tPen\WObj:=wPaper;
    MoveL Offs(pOrigin,142.04,127.88,0.00),v60,z0,tPen\WObj:=wPaper;
    MoveL Offs(pOrigin,142.04,124.28,0.00),v40,z0,tPen\WObj:=wPaper;
    MoveL Offs(pOrigin,140.98,124.28,0.00),v40,z0,tPen\WObj:=wPaper;
    MoveL Offs(pOrigin,140.98,127.58,0.00),v40,fine,tPen\WObj:=wPaper;
    MoveL Offs(pOrigin,140.98,127.58,6.00),v60,z5,tPen\WObj:=wPaper;
    MoveL Offs(pOrigin,139.93,125.17,6.00),vTravel,z5,tPen\WObj:=wPaper;
    MoveL Offs(pOrigin,139.93,125.17,0.00),v60,z0,tPen\WObj:=wPaper;
    MoveL Offs(pOrigin,139.93,124.27,0.00),v40,fine,tPen\WObj:=wPaper;
    MoveL Offs(pOrigin,139.93,124.27,6.00),v60,z5,tPen\WObj:=wPaper;
    MoveL Offs(pOrigin,135.65,123.42,6.00),vTravel,z5,tPen\WObj:=wPaper;
    MoveL Offs(pOrigin,135.65,123.42,0.00),v60,z0,tPen\WObj:=wPaper;
    MoveL Offs(pOrigin,155.00,123.42,0.00),v40,z0,tPen\WObj:=wPaper;
    MoveL Offs(pOrigin,155.59,123.89,0.00),v40,z0,tPen\WObj:=wPaper;
    MoveL Offs(pOrigin,134.70,103.00,0.00),v40,z0,tPen\WObj:=wPaper;
    MoveL Offs(pOrigin,134.03,103.06,0.00),v40,z0,tPen\WObj:=wPaper;
    MoveL Offs(pOrigin,144.85,92.24,0.00),v40,z0,tPen\WObj:=wPaper;
    MoveL Offs(pOrigin,144.19,93.08,0.00),v40,z0,tPen\WObj:=wPaper;
    MoveL Offs(pOrigin,151.41,100.29,0.00),v40,z0,tPen\WObj:=wPaper;
    MoveL Offs(pOrigin,151.45,100.47,0.00),v40,z0,tPen\WObj:=wPaper;
    MoveL Offs(pOrigin,154.30,98.53,0.00),v40,z0,tPen\WObj:=wPaper;
    MoveL Offs(pOrigin,151.45,100.47,0.00),v40,fine,tPen\WObj:=wPaper;
    MoveL Offs(pOrigin,151.45,100.47,6.00),v60,z5,tPen\WObj:=wPaper;
    MoveL Offs(pOrigin,151.79,101.73,6.00),vTravel,z5,tPen\WObj:=wPaper;
    MoveL Offs(pOrigin,151.79,101.73,0.00),v60,z0,tPen\WObj:=wPaper;
    MoveL Offs(pOrigin,134.08,119.44,0.00),v40,fine,tPen\WObj:=wPaper;
    MoveL Offs(pOrigin,134.08,119.44,6.00),v60,z5,tPen\WObj:=wPaper;
    MoveL Offs(pOrigin,132.80,120.71,6.00),vTravel,z5,tPen\WObj:=wPaper;
    MoveL Offs(pOrigin,132.80,120.71,0.00),v60,z0,tPen\WObj:=wPaper;
    MoveL Offs(pOrigin,119.54,133.97,0.00),v40,z0,tPen\WObj:=wPaper;
    MoveL Offs(pOrigin,120.15,133.25,0.00),v40,z0,tPen\WObj:=wPaper;
    MoveL Offs(pOrigin,106.89,119.99,0.00),v40,z0,tPen\WObj:=wPaper;
    MoveL Offs(pOrigin,107.90,120.25,0.00),v40,z0,tPen\WObj:=wPaper;
    MoveL Offs(pOrigin,131.30,120.25,0.00),v40,z0,tPen\WObj:=wPaper;
    MoveL Offs(pOrigin,131.15,119.19,0.00),v40,z0,tPen\WObj:=wPaper;
    MoveL Offs(pOrigin,107.90,119.19,0.00),v40,z0,tPen\WObj:=wPaper;
    MoveL Offs(pOrigin,107.90,118.14,0.00),v40,z0,tPen\WObj:=wPaper;
    MoveL Offs(pOrigin,131.15,118.14,0.00),v40,fine,tPen\WObj:=wPaper;
    MoveL Offs(pOrigin,131.15,118.14,6.00),v60,z5,tPen\WObj:=wPaper;
    MoveL Offs(pOrigin,132.11,116.83,6.00),vTravel,z5,tPen\WObj:=wPaper;
    MoveL Offs(pOrigin,132.11,116.83,0.00),v60,z0,tPen\WObj:=wPaper;
    MoveL Offs(pOrigin,108.14,92.86,0.00),v40,fine,tPen\WObj:=wPaper;
    MoveL Offs(pOrigin,108.14,92.86,6.00),v60,z5,tPen\WObj:=wPaper;
    MoveL Offs(pOrigin,109.62,92.86,6.00),vTravel,z5,tPen\WObj:=wPaper;
    MoveL Offs(pOrigin,109.62,92.86,0.00),v60,z0,tPen\WObj:=wPaper;
    MoveL Offs(pOrigin,131.79,115.03,0.00),v40,z0,tPen\WObj:=wPaper;
    MoveL Offs(pOrigin,132.79,114.76,0.00),v40,z0,tPen\WObj:=wPaper;
    MoveL Offs(pOrigin,113.38,134.17,0.00),v40,fine,tPen\WObj:=wPaper;
    MoveL Offs(pOrigin,113.38,134.17,6.00),v60,z5,tPen\WObj:=wPaper;
    MoveL Offs(pOrigin,114.30,133.37,6.00),vTravel,z5,tPen\WObj:=wPaper;
    MoveL Offs(pOrigin,114.30,133.37,0.00),v60,z0,tPen\WObj:=wPaper;
    MoveL Offs(pOrigin,106.87,125.95,0.00),v40,z0,tPen\WObj:=wPaper;
    MoveL Offs(pOrigin,106.23,126.38,0.00),v40,z0,tPen\WObj:=wPaper;
    MoveL Offs(pOrigin,132.85,99.76,0.00),v40,z0,tPen\WObj:=wPaper;
    MoveL Offs(pOrigin,133.70,100.40,0.00),v40,z0,tPen\WObj:=wPaper;
    MoveL Offs(pOrigin,141.76,92.34,0.00),v40,z0,tPen\WObj:=wPaper;
    MoveL Offs(pOrigin,141.22,93.09,0.00),v40,z0,tPen\WObj:=wPaper;
    MoveL Offs(pOrigin,155.96,107.83,0.00),v40,z0,tPen\WObj:=wPaper;
  ENDPROC

  PROC DrawPart21()
    MoveL Offs(pOrigin,156.38,107.59,0.00),v40,z0,tPen\WObj:=wPaper;
    MoveL Offs(pOrigin,129.76,134.21,0.00),v40,fine,tPen\WObj:=wPaper;
    MoveL Offs(pOrigin,129.76,134.21,6.00),v60,z5,tPen\WObj:=wPaper;
    MoveL Offs(pOrigin,131.30,131.86,6.00),vTravel,z5,tPen\WObj:=wPaper;
    MoveL Offs(pOrigin,131.30,131.86,0.00),v60,z0,tPen\WObj:=wPaper;
    MoveL Offs(pOrigin,108.05,131.86,0.00),v40,z0,tPen\WObj:=wPaper;
    MoveL Offs(pOrigin,107.90,130.81,0.00),v40,z0,tPen\WObj:=wPaper;
    MoveL Offs(pOrigin,131.45,130.81,0.00),v40,z0,tPen\WObj:=wPaper;
    MoveL Offs(pOrigin,132.39,130.56,0.00),v40,z0,tPen\WObj:=wPaper;
    MoveL Offs(pOrigin,106.93,105.10,0.00),v40,z0,tPen\WObj:=wPaper;
    MoveL Offs(pOrigin,106.17,105.53,0.00),v40,z0,tPen\WObj:=wPaper;
    MoveL Offs(pOrigin,119.64,92.06,0.00),v40,fine,tPen\WObj:=wPaper;
    MoveL Offs(pOrigin,119.64,92.06,6.00),v60,z5,tPen\WObj:=wPaper;
    MoveL Offs(pOrigin,117.72,90.50,6.00),vTravel,z5,tPen\WObj:=wPaper;
    MoveL Offs(pOrigin,117.72,90.50,0.00),v60,z0,tPen\WObj:=wPaper;
    MoveL Offs(pOrigin,106.90,79.68,0.00),v40,fine,tPen\WObj:=wPaper;
    MoveL Offs(pOrigin,106.90,79.68,6.00),v60,z5,tPen\WObj:=wPaper;
    MoveL Offs(pOrigin,105.88,78.94,6.00),vTravel,z5,tPen\WObj:=wPaper;
    MoveL Offs(pOrigin,105.88,78.94,0.00),v60,z0,tPen\WObj:=wPaper;
    MoveL Offs(pOrigin,134.83,49.98,0.00),v40,fine,tPen\WObj:=wPaper;
    MoveL Offs(pOrigin,134.83,49.98,6.00),v60,z5,tPen\WObj:=wPaper;
    MoveL Offs(pOrigin,136.23,50.77,6.00),vTravel,z5,tPen\WObj:=wPaper;
    MoveL Offs(pOrigin,136.23,50.77,0.00),v60,z0,tPen\WObj:=wPaper;
    MoveL Offs(pOrigin,164.87,79.41,0.00),v40,z0,tPen\WObj:=wPaper;
    MoveL Offs(pOrigin,164.00,79.06,0.00),v40,z0,tPen\WObj:=wPaper;
    MoveL Offs(pOrigin,135.80,79.06,0.00),v40,z0,tPen\WObj:=wPaper;
    MoveL Offs(pOrigin,135.80,80.12,0.00),v40,z0,tPen\WObj:=wPaper;
    MoveL Offs(pOrigin,164.00,80.12,0.00),v40,z0,tPen\WObj:=wPaper;
    MoveL Offs(pOrigin,163.85,81.18,0.00),v40,z0,tPen\WObj:=wPaper;
    MoveL Offs(pOrigin,135.80,81.18,0.00),v40,z0,tPen\WObj:=wPaper;
    MoveL Offs(pOrigin,135.80,82.23,0.00),v40,z0,tPen\WObj:=wPaper;
    MoveL Offs(pOrigin,163.70,82.23,0.00),v40,fine,tPen\WObj:=wPaper;
    MoveL Offs(pOrigin,163.70,82.23,6.00),v60,z5,tPen\WObj:=wPaper;
    MoveL Offs(pOrigin,165.56,81.98,6.00),vTravel,z5,tPen\WObj:=wPaper;
    MoveL Offs(pOrigin,165.56,81.98,0.00),v60,z0,tPen\WObj:=wPaper;
    MoveL Offs(pOrigin,156.33,91.21,0.00),v40,z0,tPen\WObj:=wPaper;
    MoveL Offs(pOrigin,156.65,90.60,0.00),v40,z0,tPen\WObj:=wPaper;
    MoveL Offs(pOrigin,134.80,68.75,0.00),v40,z0,tPen\WObj:=wPaper;
    MoveL Offs(pOrigin,134.14,68.60,0.00),v40,z0,tPen\WObj:=wPaper;
    MoveL Offs(pOrigin,150.26,52.47,0.00),v40,fine,tPen\WObj:=wPaper;
    MoveL Offs(pOrigin,150.26,52.47,6.00),v60,z5,tPen\WObj:=wPaper;
    MoveL Offs(pOrigin,149.45,53.72,6.00),vTravel,z5,tPen\WObj:=wPaper;
    MoveL Offs(pOrigin,149.45,53.72,0.00),v60,z0,tPen\WObj:=wPaper;
    MoveL Offs(pOrigin,135.50,53.72,0.00),v40,z0,tPen\WObj:=wPaper;
    MoveL Offs(pOrigin,135.50,54.78,0.00),v40,z0,tPen\WObj:=wPaper;
    MoveL Offs(pOrigin,151.40,54.78,0.00),v40,fine,tPen\WObj:=wPaper;
    MoveL Offs(pOrigin,151.40,54.78,6.00),v60,z5,tPen\WObj:=wPaper;
    MoveL Offs(pOrigin,153.05,55.83,6.00),vTravel,z5,tPen\WObj:=wPaper;
    MoveL Offs(pOrigin,153.05,55.83,0.00),v60,z0,tPen\WObj:=wPaper;
    MoveL Offs(pOrigin,135.50,55.83,0.00),v40,z0,tPen\WObj:=wPaper;
    MoveL Offs(pOrigin,135.50,56.89,0.00),v40,z0,tPen\WObj:=wPaper;
    MoveL Offs(pOrigin,154.40,56.89,0.00),v40,fine,tPen\WObj:=wPaper;
    MoveL Offs(pOrigin,154.40,56.89,6.00),v60,z5,tPen\WObj:=wPaper;
    MoveL Offs(pOrigin,157.41,57.28,6.00),vTravel,z5,tPen\WObj:=wPaper;
    MoveL Offs(pOrigin,157.41,57.28,0.00),v60,z0,tPen\WObj:=wPaper;
    MoveL Offs(pOrigin,134.07,80.62,0.00),v40,z0,tPen\WObj:=wPaper;
    MoveL Offs(pOrigin,134.76,80.66,0.00),v40,z0,tPen\WObj:=wPaper;
    MoveL Offs(pOrigin,144.63,90.53,0.00),v40,z0,tPen\WObj:=wPaper;
    MoveL Offs(pOrigin,144.52,91.07,0.00),v40,z0,tPen\WObj:=wPaper;
    MoveL Offs(pOrigin,165.10,70.49,0.00),v40,fine,tPen\WObj:=wPaper;
    MoveL Offs(pOrigin,165.10,70.49,6.00),v60,z5,tPen\WObj:=wPaper;
    MoveL Offs(pOrigin,164.78,69.32,6.00),vTravel,z5,tPen\WObj:=wPaper;
    MoveL Offs(pOrigin,164.78,69.32,0.00),v60,z0,tPen\WObj:=wPaper;
    MoveL Offs(pOrigin,143.04,91.06,0.00),v40,z0,tPen\WObj:=wPaper;
    MoveL Offs(pOrigin,143.03,90.42,0.00),v40,z0,tPen\WObj:=wPaper;
    MoveL Offs(pOrigin,134.86,82.26,0.00),v40,z0,tPen\WObj:=wPaper;
    MoveL Offs(pOrigin,134.18,82.00,0.00),v40,z0,tPen\WObj:=wPaper;
    MoveL Offs(pOrigin,158.15,58.03,0.00),v40,z0,tPen\WObj:=wPaper;
    MoveL Offs(pOrigin,157.85,58.88,0.00),v40,z0,tPen\WObj:=wPaper;
    MoveL Offs(pOrigin,158.75,59.78,0.00),v40,z0,tPen\WObj:=wPaper;
    MoveL Offs(pOrigin,157.85,58.88,0.00),v40,z0,tPen\WObj:=wPaper;
    MoveL Offs(pOrigin,158.90,58.77,0.00),v40,z0,tPen\WObj:=wPaper;
    MoveL Offs(pOrigin,134.19,83.49,0.00),v40,fine,tPen\WObj:=wPaper;
    MoveL Offs(pOrigin,134.19,83.49,6.00),v60,z5,tPen\WObj:=wPaper;
    MoveL Offs(pOrigin,135.80,78.01,6.00),vTravel,z5,tPen\WObj:=wPaper;
    MoveL Offs(pOrigin,135.80,78.01,0.00),v60,z0,tPen\WObj:=wPaper;
    MoveL Offs(pOrigin,164.15,78.01,0.00),v40,fine,tPen\WObj:=wPaper;
    MoveL Offs(pOrigin,164.15,78.01,6.00),v60,z5,tPen\WObj:=wPaper;
    MoveL Offs(pOrigin,164.00,73.78,6.00),vTravel,z5,tPen\WObj:=wPaper;
    MoveL Offs(pOrigin,164.00,73.78,0.00),v60,z0,tPen\WObj:=wPaper;
    MoveL Offs(pOrigin,135.80,73.78,0.00),v40,z0,tPen\WObj:=wPaper;
    MoveL Offs(pOrigin,135.80,72.73,0.00),v40,z0,tPen\WObj:=wPaper;
    MoveL Offs(pOrigin,163.70,72.73,0.00),v40,fine,tPen\WObj:=wPaper;
    MoveL Offs(pOrigin,163.70,72.73,6.00),v60,z5,tPen\WObj:=wPaper;
    MoveL Offs(pOrigin,162.65,68.50,6.00),vTravel,z5,tPen\WObj:=wPaper;
    MoveL Offs(pOrigin,162.65,68.50,0.00),v60,z0,tPen\WObj:=wPaper;
    MoveL Offs(pOrigin,135.95,68.50,0.00),v40,z0,tPen\WObj:=wPaper;
    MoveL Offs(pOrigin,135.80,67.45,0.00),v40,z0,tPen\WObj:=wPaper;
    MoveL Offs(pOrigin,162.35,67.45,0.00),v40,z0,tPen\WObj:=wPaper;
    MoveL Offs(pOrigin,161.90,66.39,0.00),v40,z0,tPen\WObj:=wPaper;
    MoveL Offs(pOrigin,135.80,66.39,0.00),v40,z0,tPen\WObj:=wPaper;
    MoveL Offs(pOrigin,135.80,65.34,0.00),v40,z0,tPen\WObj:=wPaper;
    MoveL Offs(pOrigin,161.45,65.34,0.00),v40,fine,tPen\WObj:=wPaper;
    MoveL Offs(pOrigin,161.45,65.34,6.00),v60,z5,tPen\WObj:=wPaper;
    MoveL Offs(pOrigin,156.80,59.00,6.00),vTravel,z5,tPen\WObj:=wPaper;
    MoveL Offs(pOrigin,156.80,59.00,0.00),v60,z0,tPen\WObj:=wPaper;
    MoveL Offs(pOrigin,135.50,59.00,0.00),v40,fine,tPen\WObj:=wPaper;
    MoveL Offs(pOrigin,135.50,59.00,6.00),v60,z5,tPen\WObj:=wPaper;
    MoveL Offs(pOrigin,133.79,58.49,6.00),vTravel,z5,tPen\WObj:=wPaper;
    MoveL Offs(pOrigin,133.79,58.49,0.00),v60,z0,tPen\WObj:=wPaper;
    MoveL Offs(pOrigin,142.28,50.00,0.00),v40,fine,tPen\WObj:=wPaper;
    MoveL Offs(pOrigin,142.28,50.00,6.00),v60,z5,tPen\WObj:=wPaper;
    MoveL Offs(pOrigin,136.75,49.56,6.00),vTravel,z5,tPen\WObj:=wPaper;
    MoveL Offs(pOrigin,136.75,49.56,0.00),v60,z0,tPen\WObj:=wPaper;
    MoveL Offs(pOrigin,105.78,80.53,0.00),v40,fine,tPen\WObj:=wPaper;
    MoveL Offs(pOrigin,105.78,80.53,6.00),v60,z5,tPen\WObj:=wPaper;
    MoveL Offs(pOrigin,106.21,83.09,6.00),vTravel,z5,tPen\WObj:=wPaper;
    MoveL Offs(pOrigin,106.21,83.09,0.00),v60,z0,tPen\WObj:=wPaper;
    MoveL Offs(pOrigin,132.83,56.47,0.00),v40,fine,tPen\WObj:=wPaper;
    MoveL Offs(pOrigin,132.83,56.47,6.00),v60,z5,tPen\WObj:=wPaper;
    MoveL Offs(pOrigin,132.94,57.85,6.00),vTravel,z5,tPen\WObj:=wPaper;
    MoveL Offs(pOrigin,132.94,57.85,0.00),v60,z0,tPen\WObj:=wPaper;
    MoveL Offs(pOrigin,106.21,84.58,0.00),v40,fine,tPen\WObj:=wPaper;
    MoveL Offs(pOrigin,106.21,84.58,6.00),v60,z5,tPen\WObj:=wPaper;
    MoveL Offs(pOrigin,108.35,89.62,6.00),vTravel,z5,tPen\WObj:=wPaper;
    MoveL Offs(pOrigin,108.35,89.62,0.00),v60,z0,tPen\WObj:=wPaper;
    MoveL Offs(pOrigin,124.40,89.62,0.00),v40,z0,tPen\WObj:=wPaper;
    MoveL Offs(pOrigin,123.67,90.48,0.00),v40,z0,tPen\WObj:=wPaper;
    MoveL Offs(pOrigin,106.91,73.72,0.00),v40,z0,tPen\WObj:=wPaper;
    MoveL Offs(pOrigin,107.90,73.78,0.00),v40,z0,tPen\WObj:=wPaper;
  ENDPROC

  PROC DrawPart22()
    MoveL Offs(pOrigin,131.00,73.78,0.00),v40,z0,tPen\WObj:=wPaper;
    MoveL Offs(pOrigin,131.81,73.22,0.00),v40,z0,tPen\WObj:=wPaper;
    MoveL Offs(pOrigin,109.32,50.74,0.00),v40,fine,tPen\WObj:=wPaper;
    MoveL Offs(pOrigin,109.32,50.74,6.00),v60,z5,tPen\WObj:=wPaper;
    MoveL Offs(pOrigin,109.84,49.59,6.00),vTravel,z5,tPen\WObj:=wPaper;
    MoveL Offs(pOrigin,109.84,49.59,0.00),v60,z0,tPen\WObj:=wPaper;
    MoveL Offs(pOrigin,105.91,53.52,0.00),v40,fine,tPen\WObj:=wPaper;
    MoveL Offs(pOrigin,105.91,53.52,6.00),v60,z5,tPen\WObj:=wPaper;
    MoveL Offs(pOrigin,105.59,52.35,6.00),vTravel,z5,tPen\WObj:=wPaper;
    MoveL Offs(pOrigin,105.59,52.35,0.00),v60,z0,tPen\WObj:=wPaper;
    MoveL Offs(pOrigin,108.56,49.38,0.00),v40,fine,tPen\WObj:=wPaper;
    MoveL Offs(pOrigin,108.56,49.38,6.00),v60,z5,tPen\WObj:=wPaper;
    MoveL Offs(pOrigin,107.08,51.49,6.00),vTravel,z5,tPen\WObj:=wPaper;
    MoveL Offs(pOrigin,107.08,51.49,0.00),v60,z0,tPen\WObj:=wPaper;
    MoveL Offs(pOrigin,131.80,76.20,0.00),v40,z0,tPen\WObj:=wPaper;
    MoveL Offs(pOrigin,132.46,76.25,0.00),v40,z0,tPen\WObj:=wPaper;
    MoveL Offs(pOrigin,106.05,102.66,0.00),v40,fine,tPen\WObj:=wPaper;
    MoveL Offs(pOrigin,106.05,102.66,6.00),v60,z5,tPen\WObj:=wPaper;
    MoveL Offs(pOrigin,105.73,101.49,6.00),vTravel,z5,tPen\WObj:=wPaper;
    MoveL Offs(pOrigin,105.73,101.49,0.00),v60,z0,tPen\WObj:=wPaper;
    MoveL Offs(pOrigin,132.56,74.65,0.00),v40,fine,tPen\WObj:=wPaper;
    MoveL Offs(pOrigin,132.56,74.65,6.00),v60,z5,tPen\WObj:=wPaper;
    MoveL Offs(pOrigin,132.77,72.95,6.00),vTravel,z5,tPen\WObj:=wPaper;
    MoveL Offs(pOrigin,132.77,72.95,0.00),v60,z0,tPen\WObj:=wPaper;
    MoveL Offs(pOrigin,105.83,99.89,0.00),v40,fine,tPen\WObj:=wPaper;
    MoveL Offs(pOrigin,105.83,99.89,6.00),v60,z5,tPen\WObj:=wPaper;
    MoveL Offs(pOrigin,107.75,101.24,6.00),vTravel,z5,tPen\WObj:=wPaper;
    MoveL Offs(pOrigin,107.75,101.24,0.00),v60,z0,tPen\WObj:=wPaper;
    MoveL Offs(pOrigin,131.45,101.24,0.00),v40,fine,tPen\WObj:=wPaper;
    MoveL Offs(pOrigin,131.45,101.24,6.00),v60,z5,tPen\WObj:=wPaper;
    MoveL Offs(pOrigin,132.85,101.25,6.00),vTravel,z5,tPen\WObj:=wPaper;
    MoveL Offs(pOrigin,132.85,101.25,0.00),v60,z0,tPen\WObj:=wPaper;
    MoveL Offs(pOrigin,105.70,128.40,0.00),v40,fine,tPen\WObj:=wPaper;
    MoveL Offs(pOrigin,105.70,128.40,6.00),v60,z5,tPen\WObj:=wPaper;
    MoveL Offs(pOrigin,105.70,129.89,6.00),vTravel,z5,tPen\WObj:=wPaper;
    MoveL Offs(pOrigin,105.70,129.89,0.00),v60,z0,tPen\WObj:=wPaper;
    MoveL Offs(pOrigin,132.54,103.05,0.00),v40,fine,tPen\WObj:=wPaper;
    MoveL Offs(pOrigin,132.54,103.05,6.00),v60,z5,tPen\WObj:=wPaper;
    MoveL Offs(pOrigin,131.30,104.41,6.00),vTravel,z5,tPen\WObj:=wPaper;
    MoveL Offs(pOrigin,131.30,104.41,0.00),v60,z0,tPen\WObj:=wPaper;
    MoveL Offs(pOrigin,107.90,104.41,0.00),v40,z0,tPen\WObj:=wPaper;
    MoveL Offs(pOrigin,107.90,105.46,0.00),v40,z0,tPen\WObj:=wPaper;
    MoveL Offs(pOrigin,131.30,105.46,0.00),v40,z0,tPen\WObj:=wPaper;
    MoveL Offs(pOrigin,131.30,106.52,0.00),v40,z0,tPen\WObj:=wPaper;
    MoveL Offs(pOrigin,107.75,106.52,0.00),v40,z0,tPen\WObj:=wPaper;
    MoveL Offs(pOrigin,106.93,106.59,0.00),v40,z0,tPen\WObj:=wPaper;
    MoveL Offs(pOrigin,132.17,131.83,0.00),v40,fine,tPen\WObj:=wPaper;
    MoveL Offs(pOrigin,132.17,131.83,6.00),v60,z5,tPen\WObj:=wPaper;
    MoveL Offs(pOrigin,131.45,129.75,6.00),vTravel,z5,tPen\WObj:=wPaper;
    MoveL Offs(pOrigin,131.45,129.75,0.00),v60,z0,tPen\WObj:=wPaper;
    MoveL Offs(pOrigin,107.90,129.75,0.00),v40,fine,tPen\WObj:=wPaper;
    MoveL Offs(pOrigin,107.90,129.75,6.00),v60,z5,tPen\WObj:=wPaper;
    MoveL Offs(pOrigin,106.67,133.40,6.00),vTravel,z5,tPen\WObj:=wPaper;
    MoveL Offs(pOrigin,106.67,133.40,0.00),v60,z0,tPen\WObj:=wPaper;
    MoveL Offs(pOrigin,132.76,107.31,0.00),v40,fine,tPen\WObj:=wPaper;
    MoveL Offs(pOrigin,132.76,107.31,6.00),v60,z5,tPen\WObj:=wPaper;
    MoveL Offs(pOrigin,129.37,105.82,6.00),vTravel,z5,tPen\WObj:=wPaper;
    MoveL Offs(pOrigin,129.37,105.82,0.00),v60,z0,tPen\WObj:=wPaper;
    MoveL Offs(pOrigin,129.37,95.32,0.00),v40,fine,tPen\WObj:=wPaper;
    MoveL Offs(pOrigin,129.37,95.32,6.00),v60,z5,tPen\WObj:=wPaper;
    MoveL Offs(pOrigin,131.30,95.96,6.00),vTravel,z5,tPen\WObj:=wPaper;
    MoveL Offs(pOrigin,131.30,95.96,0.00),v60,z0,tPen\WObj:=wPaper;
    MoveL Offs(pOrigin,107.75,95.96,0.00),v40,fine,tPen\WObj:=wPaper;
    MoveL Offs(pOrigin,107.75,95.96,6.00),v60,z5,tPen\WObj:=wPaper;
    MoveL Offs(pOrigin,106.03,95.21,6.00),vTravel,z5,tPen\WObj:=wPaper;
    MoveL Offs(pOrigin,106.03,95.21,0.00),v60,z0,tPen\WObj:=wPaper;
    MoveL Offs(pOrigin,132.44,68.80,0.00),v40,z0,tPen\WObj:=wPaper;
    MoveL Offs(pOrigin,131.82,68.76,0.00),v40,z0,tPen\WObj:=wPaper;
    MoveL Offs(pOrigin,113.79,50.73,0.00),v40,fine,tPen\WObj:=wPaper;
    MoveL Offs(pOrigin,113.79,50.73,6.00),v60,z5,tPen\WObj:=wPaper;
    MoveL Offs(pOrigin,114.41,49.50,6.00),vTravel,z5,tPen\WObj:=wPaper;
    MoveL Offs(pOrigin,114.41,49.50,0.00),v60,z0,tPen\WObj:=wPaper;
    MoveL Offs(pOrigin,105.71,58.20,0.00),v40,fine,tPen\WObj:=wPaper;
    MoveL Offs(pOrigin,105.71,58.20,6.00),v60,z5,tPen\WObj:=wPaper;
    MoveL Offs(pOrigin,107.90,57.94,6.00),vTravel,z5,tPen\WObj:=wPaper;
    MoveL Offs(pOrigin,107.90,57.94,0.00),v60,z0,tPen\WObj:=wPaper;
    MoveL Offs(pOrigin,131.15,57.94,0.00),v40,fine,tPen\WObj:=wPaper;
    MoveL Offs(pOrigin,131.15,57.94,6.00),v60,z5,tPen\WObj:=wPaper;
    MoveL Offs(pOrigin,131.30,55.83,6.00),vTravel,z5,tPen\WObj:=wPaper;
    MoveL Offs(pOrigin,131.30,55.83,0.00),v60,z0,tPen\WObj:=wPaper;
    MoveL Offs(pOrigin,107.90,55.83,0.00),v40,z0,tPen\WObj:=wPaper;
    MoveL Offs(pOrigin,107.90,54.78,0.00),v40,z0,tPen\WObj:=wPaper;
    MoveL Offs(pOrigin,131.30,54.78,0.00),v40,z0,tPen\WObj:=wPaper;
    MoveL Offs(pOrigin,131.30,53.72,0.00),v40,z0,tPen\WObj:=wPaper;
    MoveL Offs(pOrigin,107.75,53.72,0.00),v40,fine,tPen\WObj:=wPaper;
    MoveL Offs(pOrigin,107.75,53.72,6.00),v60,z5,tPen\WObj:=wPaper;
    MoveL Offs(pOrigin,107.90,68.50,6.00),vTravel,z5,tPen\WObj:=wPaper;
    MoveL Offs(pOrigin,107.90,68.50,0.00),v60,z0,tPen\WObj:=wPaper;
    MoveL Offs(pOrigin,131.15,68.50,0.00),v40,z0,tPen\WObj:=wPaper;
    MoveL Offs(pOrigin,131.00,69.56,0.00),v40,z0,tPen\WObj:=wPaper;
    MoveL Offs(pOrigin,107.90,69.56,0.00),v40,fine,tPen\WObj:=wPaper;
    MoveL Offs(pOrigin,107.90,69.56,6.00),v60,z5,tPen\WObj:=wPaper;
    MoveL Offs(pOrigin,107.90,71.67,6.00),vTravel,z5,tPen\WObj:=wPaper;
    MoveL Offs(pOrigin,107.90,71.67,0.00),v60,z0,tPen\WObj:=wPaper;
    MoveL Offs(pOrigin,131.15,71.67,0.00),v40,z0,tPen\WObj:=wPaper;
    MoveL Offs(pOrigin,131.15,72.73,0.00),v40,z0,tPen\WObj:=wPaper;
    MoveL Offs(pOrigin,107.90,72.73,0.00),v40,fine,tPen\WObj:=wPaper;
    MoveL Offs(pOrigin,107.90,72.73,6.00),v60,z5,tPen\WObj:=wPaper;
    MoveL Offs(pOrigin,105.54,73.30,6.00),vTravel,z5,tPen\WObj:=wPaper;
    MoveL Offs(pOrigin,105.54,73.30,0.00),v60,z0,tPen\WObj:=wPaper;
    MoveL Offs(pOrigin,129.51,49.33,0.00),v40,fine,tPen\WObj:=wPaper;
    MoveL Offs(pOrigin,129.51,49.33,6.00),v60,z5,tPen\WObj:=wPaper;
    MoveL Offs(pOrigin,130.69,49.65,6.00),vTravel,z5,tPen\WObj:=wPaper;
    MoveL Offs(pOrigin,130.69,49.65,0.00),v60,z0,tPen\WObj:=wPaper;
    MoveL Offs(pOrigin,105.87,74.47,0.00),v40,fine,tPen\WObj:=wPaper;
    MoveL Offs(pOrigin,105.87,74.47,6.00),v60,z5,tPen\WObj:=wPaper;
    MoveL Offs(pOrigin,106.19,75.64,6.00),vTravel,z5,tPen\WObj:=wPaper;
    MoveL Offs(pOrigin,106.19,75.64,0.00),v60,z0,tPen\WObj:=wPaper;
    MoveL Offs(pOrigin,131.86,49.97,0.00),v40,z0,tPen\WObj:=wPaper;
    MoveL Offs(pOrigin,132.71,50.62,0.00),v40,z0,tPen\WObj:=wPaper;
    MoveL Offs(pOrigin,106.19,77.13,0.00),v40,fine,tPen\WObj:=wPaper;
    MoveL Offs(pOrigin,106.19,77.13,6.00),v60,z5,tPen\WObj:=wPaper;
    MoveL Offs(pOrigin,106.91,75.21,6.00),vTravel,z5,tPen\WObj:=wPaper;
    MoveL Offs(pOrigin,106.91,75.21,0.00),v60,z0,tPen\WObj:=wPaper;
    MoveL Offs(pOrigin,122.29,90.59,0.00),v40,fine,tPen\WObj:=wPaper;
    MoveL Offs(pOrigin,122.29,90.59,6.00),v60,z5,tPen\WObj:=wPaper;
    MoveL Offs(pOrigin,131.23,92.41,6.00),vTravel,z5,tPen\WObj:=wPaper;
    MoveL Offs(pOrigin,131.23,92.41,0.00),v60,z0,tPen\WObj:=wPaper;
    MoveL Offs(pOrigin,106.09,117.55,0.00),v40,fine,tPen\WObj:=wPaper;
    MoveL Offs(pOrigin,106.09,117.55,6.00),v60,z5,tPen\WObj:=wPaper;
  ENDPROC

  PROC DrawPart23()
    MoveL Offs(pOrigin,106.89,118.50,6.00),vTravel,z5,tPen\WObj:=wPaper;
    MoveL Offs(pOrigin,106.89,118.50,0.00),v60,z0,tPen\WObj:=wPaper;
    MoveL Offs(pOrigin,121.74,133.35,0.00),v40,z0,tPen\WObj:=wPaper;
    MoveL Offs(pOrigin,122.31,134.19,0.00),v40,z0,tPen\WObj:=wPaper;
    MoveL Offs(pOrigin,153.28,103.22,0.00),v40,z0,tPen\WObj:=wPaper;
    MoveL Offs(pOrigin,152.90,103.43,0.00),v40,z0,tPen\WObj:=wPaper;
    MoveL Offs(pOrigin,153.50,104.03,0.00),v40,z0,tPen\WObj:=wPaper;
    MoveL Offs(pOrigin,152.90,103.43,0.00),v40,z0,tPen\WObj:=wPaper;
    MoveL Offs(pOrigin,152.53,102.47,0.00),v40,z0,tPen\WObj:=wPaper;
    MoveL Offs(pOrigin,120.82,134.19,0.00),v40,fine,tPen\WObj:=wPaper;
    MoveL Offs(pOrigin,120.82,134.19,6.00),v60,z5,tPen\WObj:=wPaper;
    MoveL Offs(pOrigin,120.92,130.88,6.00),vTravel,z5,tPen\WObj:=wPaper;
    MoveL Offs(pOrigin,120.92,130.88,0.00),v60,z0,tPen\WObj:=wPaper;
    MoveL Offs(pOrigin,120.92,127.87,0.00),v40,z0,tPen\WObj:=wPaper;
    MoveL Offs(pOrigin,121.98,127.57,0.00),v40,z0,tPen\WObj:=wPaper;
    MoveL Offs(pOrigin,121.98,131.02,0.00),v40,z0,tPen\WObj:=wPaper;
    MoveL Offs(pOrigin,123.03,131.02,0.00),v40,z0,tPen\WObj:=wPaper;
    MoveL Offs(pOrigin,123.03,127.87,0.00),v40,fine,tPen\WObj:=wPaper;
    MoveL Offs(pOrigin,123.03,127.87,6.00),v60,z5,tPen\WObj:=wPaper;
    MoveL Offs(pOrigin,124.09,129.07,6.00),vTravel,z5,tPen\WObj:=wPaper;
    MoveL Offs(pOrigin,124.09,129.07,0.00),v60,z0,tPen\WObj:=wPaper;
    MoveL Offs(pOrigin,124.09,131.32,0.00),v40,z0,tPen\WObj:=wPaper;
    MoveL Offs(pOrigin,125.14,131.32,0.00),v40,z0,tPen\WObj:=wPaper;
    MoveL Offs(pOrigin,125.14,129.82,0.00),v40,z0,tPen\WObj:=wPaper;
    MoveL Offs(pOrigin,126.20,130.27,0.00),v40,z0,tPen\WObj:=wPaper;
    MoveL Offs(pOrigin,126.20,131.17,0.00),v40,fine,tPen\WObj:=wPaper;
    MoveL Offs(pOrigin,126.20,131.17,6.00),v60,z5,tPen\WObj:=wPaper;
    MoveL Offs(pOrigin,124.72,133.34,6.00),vTravel,z5,tPen\WObj:=wPaper;
    MoveL Offs(pOrigin,124.72,133.34,0.00),v60,z0,tPen\WObj:=wPaper;
    MoveL Offs(pOrigin,106.90,115.52,0.00),v40,fine,tPen\WObj:=wPaper;
    MoveL Offs(pOrigin,106.90,115.52,6.00),v60,z5,tPen\WObj:=wPaper;
    MoveL Offs(pOrigin,107.90,112.86,6.00),vTravel,z5,tPen\WObj:=wPaper;
    MoveL Offs(pOrigin,107.90,112.86,0.00),v60,z0,tPen\WObj:=wPaper;
    MoveL Offs(pOrigin,131.00,112.86,0.00),v40,z0,tPen\WObj:=wPaper;
    MoveL Offs(pOrigin,131.15,111.80,0.00),v40,z0,tPen\WObj:=wPaper;
    MoveL Offs(pOrigin,107.90,111.80,0.00),v40,z0,tPen\WObj:=wPaper;
    MoveL Offs(pOrigin,107.90,110.74,0.00),v40,z0,tPen\WObj:=wPaper;
    MoveL Offs(pOrigin,131.15,110.74,0.00),v40,fine,tPen\WObj:=wPaper;
    MoveL Offs(pOrigin,131.15,110.74,6.00),v60,z5,tPen\WObj:=wPaper;
    MoveL Offs(pOrigin,132.79,116.24,6.00),vTravel,z5,tPen\WObj:=wPaper;
    MoveL Offs(pOrigin,132.79,116.24,0.00),v60,z0,tPen\WObj:=wPaper;
    MoveL Offs(pOrigin,114.86,134.17,0.00),v40,fine,tPen\WObj:=wPaper;
    MoveL Offs(pOrigin,114.86,134.17,6.00),v60,z5,tPen\WObj:=wPaper;
    MoveL Offs(pOrigin,117.27,133.36,6.00),vTravel,z5,tPen\WObj:=wPaper;
    MoveL Offs(pOrigin,117.27,133.36,0.00),v60,z0,tPen\WObj:=wPaper;
    MoveL Offs(pOrigin,106.88,122.97,0.00),v40,z0,tPen\WObj:=wPaper;
    MoveL Offs(pOrigin,107.90,122.36,0.00),v40,z0,tPen\WObj:=wPaper;
    MoveL Offs(pOrigin,131.30,122.36,0.00),v40,fine,tPen\WObj:=wPaper;
    MoveL Offs(pOrigin,131.30,122.36,6.00),v60,z5,tPen\WObj:=wPaper;
    MoveL Offs(pOrigin,133.77,124.23,6.00),vTravel,z5,tPen\WObj:=wPaper;
    MoveL Offs(pOrigin,133.77,124.23,0.00),v60,z0,tPen\WObj:=wPaper;
    MoveL Offs(pOrigin,154.03,103.97,0.00),v40,fine,tPen\WObj:=wPaper;
    MoveL Offs(pOrigin,154.03,103.97,6.00),v60,z5,tPen\WObj:=wPaper;
    MoveL Offs(pOrigin,152.60,104.41,6.00),vTravel,z5,tPen\WObj:=wPaper;
    MoveL Offs(pOrigin,152.60,104.41,0.00),v60,z0,tPen\WObj:=wPaper;
    MoveL Offs(pOrigin,135.50,104.41,0.00),v40,z0,tPen\WObj:=wPaper;
    MoveL Offs(pOrigin,135.50,103.35,0.00),v40,z0,tPen\WObj:=wPaper;
    MoveL Offs(pOrigin,151.55,103.35,0.00),v40,fine,tPen\WObj:=wPaper;
    MoveL Offs(pOrigin,151.55,103.35,6.00),v60,z5,tPen\WObj:=wPaper;
    MoveL Offs(pOrigin,147.32,102.52,6.00),vTravel,z5,tPen\WObj:=wPaper;
    MoveL Offs(pOrigin,147.32,102.52,0.00),v60,z0,tPen\WObj:=wPaper;
    MoveL Offs(pOrigin,147.32,94.87,0.00),v40,fine,tPen\WObj:=wPaper;
    MoveL Offs(pOrigin,147.32,94.87,6.00),v60,z5,tPen\WObj:=wPaper;
    MoveL Offs(pOrigin,146.26,96.67,6.00),vTravel,z5,tPen\WObj:=wPaper;
    MoveL Offs(pOrigin,146.26,96.67,0.00),v60,z0,tPen\WObj:=wPaper;
    MoveL Offs(pOrigin,146.26,102.52,0.00),v40,z0,tPen\WObj:=wPaper;
    MoveL Offs(pOrigin,145.21,102.82,0.00),v40,z0,tPen\WObj:=wPaper;
    MoveL Offs(pOrigin,145.21,96.52,0.00),v40,z0,tPen\WObj:=wPaper;
    MoveL Offs(pOrigin,144.15,96.52,0.00),v40,z0,tPen\WObj:=wPaper;
    MoveL Offs(pOrigin,144.15,106.12,0.00),v40,z0,tPen\WObj:=wPaper;
    MoveL Offs(pOrigin,143.10,105.98,0.00),v40,z0,tPen\WObj:=wPaper;
    MoveL Offs(pOrigin,143.10,95.62,0.00),v40,fine,tPen\WObj:=wPaper;
    MoveL Offs(pOrigin,143.10,95.62,6.00),v60,z5,tPen\WObj:=wPaper;
    MoveL Offs(pOrigin,142.04,95.02,6.00),vTravel,z5,tPen\WObj:=wPaper;
    MoveL Offs(pOrigin,142.04,95.02,0.00),v60,z0,tPen\WObj:=wPaper;
    MoveL Offs(pOrigin,142.04,105.82,0.00),v40,z0,tPen\WObj:=wPaper;
    MoveL Offs(pOrigin,140.98,105.68,0.00),v40,z0,tPen\WObj:=wPaper;
    MoveL Offs(pOrigin,140.98,94.72,0.00),v40,z0,tPen\WObj:=wPaper;
    MoveL Offs(pOrigin,139.93,94.72,0.00),v40,z0,tPen\WObj:=wPaper;
    MoveL Offs(pOrigin,139.93,105.68,0.00),v40,z0,tPen\WObj:=wPaper;
    MoveL Offs(pOrigin,138.87,105.52,0.00),v40,z0,tPen\WObj:=wPaper;
    MoveL Offs(pOrigin,138.87,94.72,0.00),v40,z0,tPen\WObj:=wPaper;
    MoveL Offs(pOrigin,137.82,94.72,0.00),v40,z0,tPen\WObj:=wPaper;
    MoveL Offs(pOrigin,137.82,104.32,0.00),v40,z0,tPen\WObj:=wPaper;
    MoveL Offs(pOrigin,136.76,104.02,0.00),v40,z0,tPen\WObj:=wPaper;
    MoveL Offs(pOrigin,136.76,94.72,0.00),v40,fine,tPen\WObj:=wPaper;
    MoveL Offs(pOrigin,136.76,94.72,6.00),v60,z5,tPen\WObj:=wPaper;
    MoveL Offs(pOrigin,135.65,93.85,6.00),vTravel,z5,tPen\WObj:=wPaper;
    MoveL Offs(pOrigin,135.65,93.85,0.00),v60,z0,tPen\WObj:=wPaper;
    MoveL Offs(pOrigin,157.85,93.85,0.00),v40,z0,tPen\WObj:=wPaper;
    MoveL Offs(pOrigin,157.49,92.94,0.00),v40,z0,tPen\WObj:=wPaper;
    MoveL Offs(pOrigin,158.87,94.31,0.00),v40,fine,tPen\WObj:=wPaper;
    MoveL Offs(pOrigin,158.87,94.31,6.00),v60,z5,tPen\WObj:=wPaper;
    MoveL Offs(pOrigin,157.88,88.28,6.00),vTravel,z5,tPen\WObj:=wPaper;
    MoveL Offs(pOrigin,157.88,88.28,0.00),v60,z0,tPen\WObj:=wPaper;
    MoveL Offs(pOrigin,157.88,86.62,0.00),v40,fine,tPen\WObj:=wPaper;
    MoveL Offs(pOrigin,157.88,86.62,6.00),v60,z5,tPen\WObj:=wPaper;
    MoveL Offs(pOrigin,156.82,85.87,6.00),vTravel,z5,tPen\WObj:=wPaper;
    MoveL Offs(pOrigin,156.82,85.87,0.00),v60,z0,tPen\WObj:=wPaper;
    MoveL Offs(pOrigin,156.82,88.28,0.00),v40,z0,tPen\WObj:=wPaper;
    MoveL Offs(pOrigin,155.77,88.28,0.00),v40,z0,tPen\WObj:=wPaper;
    MoveL Offs(pOrigin,155.77,86.32,0.00),v40,z0,tPen\WObj:=wPaper;
    MoveL Offs(pOrigin,154.71,86.62,0.00),v40,z0,tPen\WObj:=wPaper;
    MoveL Offs(pOrigin,154.71,88.28,0.00),v40,z0,tPen\WObj:=wPaper;
    MoveL Offs(pOrigin,153.66,88.12,0.00),v40,z0,tPen\WObj:=wPaper;
    MoveL Offs(pOrigin,153.66,86.92,0.00),v40,fine,tPen\WObj:=wPaper;
    MoveL Offs(pOrigin,153.66,86.92,6.00),v60,z5,tPen\WObj:=wPaper;
    MoveL Offs(pOrigin,146.60,89.62,6.00),vTravel,z5,tPen\WObj:=wPaper;
    MoveL Offs(pOrigin,146.60,89.62,0.00),v60,z0,tPen\WObj:=wPaper;
    MoveL Offs(pOrigin,142.40,89.62,0.00),v40,fine,tPen\WObj:=wPaper;
    MoveL Offs(pOrigin,142.40,89.62,6.00),v60,z5,tPen\WObj:=wPaper;
    MoveL Offs(pOrigin,135.70,92.43,6.00),vTravel,z5,tPen\WObj:=wPaper;
    MoveL Offs(pOrigin,135.70,92.43,0.00),v60,z0,tPen\WObj:=wPaper;
    MoveL Offs(pOrigin,133.79,94.34,0.00),v40,z0,tPen\WObj:=wPaper;
    MoveL Offs(pOrigin,132.83,93.80,0.00),v40,z0,tPen\WObj:=wPaper;
    MoveL Offs(pOrigin,105.89,120.74,0.00),v40,fine,tPen\WObj:=wPaper;
    MoveL Offs(pOrigin,105.89,120.74,6.00),v60,z5,tPen\WObj:=wPaper;
    MoveL Offs(pOrigin,106.21,118.93,6.00),vTravel,z5,tPen\WObj:=wPaper;
    MoveL Offs(pOrigin,106.21,118.93,0.00),v60,z0,tPen\WObj:=wPaper;
    MoveL Offs(pOrigin,132.19,92.95,0.00),v40,fine,tPen\WObj:=wPaper;
  ENDPROC

  PROC DrawPart24()
    MoveL Offs(pOrigin,132.19,92.95,6.00),v60,z5,tPen\WObj:=wPaper;
    MoveL Offs(pOrigin,130.42,97.57,6.00),vTravel,z5,tPen\WObj:=wPaper;
    MoveL Offs(pOrigin,130.42,97.57,0.00),v60,z0,tPen\WObj:=wPaper;
    MoveL Offs(pOrigin,130.42,99.82,0.00),v40,fine,tPen\WObj:=wPaper;
    MoveL Offs(pOrigin,130.42,99.82,6.00),v60,z5,tPen\WObj:=wPaper;
    MoveL Offs(pOrigin,148.77,93.17,6.00),vTravel,z5,tPen\WObj:=wPaper;
    MoveL Offs(pOrigin,148.77,93.17,0.00),v60,z0,tPen\WObj:=wPaper;
    MoveL Offs(pOrigin,154.18,98.58,0.00),v40,fine,tPen\WObj:=wPaper;
    MoveL Offs(pOrigin,154.18,98.58,6.00),v60,z5,tPen\WObj:=wPaper;
    MoveL Offs(pOrigin,152.60,97.72,6.00),vTravel,z5,tPen\WObj:=wPaper;
    MoveL Offs(pOrigin,152.60,97.72,0.00),v60,z0,tPen\WObj:=wPaper;
    MoveL Offs(pOrigin,152.60,94.87,0.00),v40,z0,tPen\WObj:=wPaper;
    MoveL Offs(pOrigin,151.54,94.72,0.00),v40,z0,tPen\WObj:=wPaper;
    MoveL Offs(pOrigin,151.54,98.32,0.00),v40,fine,tPen\WObj:=wPaper;
    MoveL Offs(pOrigin,151.54,98.32,6.00),v60,z5,tPen\WObj:=wPaper;
    MoveL Offs(pOrigin,150.49,99.07,6.00),vTravel,z5,tPen\WObj:=wPaper;
    MoveL Offs(pOrigin,150.49,99.07,0.00),v60,z0,tPen\WObj:=wPaper;
    MoveL Offs(pOrigin,150.49,94.72,0.00),v40,fine,tPen\WObj:=wPaper;
    MoveL Offs(pOrigin,150.49,94.72,6.00),v60,z5,tPen\WObj:=wPaper;
    MoveL Offs(pOrigin,158.21,116.21,6.00),vTravel,z5,tPen\WObj:=wPaper;
    MoveL Offs(pOrigin,158.21,116.21,0.00),v60,z0,tPen\WObj:=wPaper;
    MoveL Offs(pOrigin,140.50,133.92,0.00),v40,z0,tPen\WObj:=wPaper;
    MoveL Offs(pOrigin,140.99,133.19,0.00),v40,z0,tPen\WObj:=wPaper;
    MoveL Offs(pOrigin,134.63,126.83,0.00),v40,z0,tPen\WObj:=wPaper;
    MoveL Offs(pOrigin,135.50,126.58,0.00),v40,z0,tPen\WObj:=wPaper;
    MoveL Offs(pOrigin,152.75,126.58,0.00),v40,fine,tPen\WObj:=wPaper;
    MoveL Offs(pOrigin,152.75,126.58,6.00),v60,z5,tPen\WObj:=wPaper;
    MoveL Offs(pOrigin,151.70,127.64,6.00),vTravel,z5,tPen\WObj:=wPaper;
    MoveL Offs(pOrigin,151.70,127.64,0.00),v60,z0,tPen\WObj:=wPaper;
    MoveL Offs(pOrigin,135.35,127.64,0.00),v40,fine,tPen\WObj:=wPaper;
    MoveL Offs(pOrigin,135.35,127.64,6.00),v60,z5,tPen\WObj:=wPaper;
    MoveL Offs(pOrigin,138.87,129.67,6.00),vTravel,z5,tPen\WObj:=wPaper;
    MoveL Offs(pOrigin,138.87,129.67,0.00),v60,z0,tPen\WObj:=wPaper;
    MoveL Offs(pOrigin,138.87,131.32,0.00),v40,fine,tPen\WObj:=wPaper;
    MoveL Offs(pOrigin,138.87,131.32,6.00),v60,z5,tPen\WObj:=wPaper;
    MoveL Offs(pOrigin,129.37,127.27,6.00),vTravel,z5,tPen\WObj:=wPaper;
    MoveL Offs(pOrigin,129.37,127.27,0.00),v60,z0,tPen\WObj:=wPaper;
    MoveL Offs(pOrigin,129.37,125.77,0.00),v40,fine,tPen\WObj:=wPaper;
    MoveL Offs(pOrigin,129.37,125.77,6.00),v60,z5,tPen\WObj:=wPaper;
    MoveL Offs(pOrigin,119.86,128.32,6.00),vTravel,z5,tPen\WObj:=wPaper;
    MoveL Offs(pOrigin,119.86,128.32,0.00),v60,z0,tPen\WObj:=wPaper;
    MoveL Offs(pOrigin,119.86,130.88,0.00),v40,fine,tPen\WObj:=wPaper;
    MoveL Offs(pOrigin,119.86,130.88,6.00),v60,z5,tPen\WObj:=wPaper;
    MoveL Offs(pOrigin,118.81,129.97,6.00),vTravel,z5,tPen\WObj:=wPaper;
    MoveL Offs(pOrigin,118.81,129.97,0.00),v60,z0,tPen\WObj:=wPaper;
    MoveL Offs(pOrigin,118.81,128.77,0.00),v40,fine,tPen\WObj:=wPaper;
    MoveL Offs(pOrigin,118.81,128.77,6.00),v60,z5,tPen\WObj:=wPaper;
    MoveL Offs(pOrigin,152.72,129.17,6.00),vTravel,z5,tPen\WObj:=wPaper;
    MoveL Offs(pOrigin,152.72,129.17,0.00),v60,z0,tPen\WObj:=wPaper;
    MoveL Offs(pOrigin,154.10,127.79,0.00),v40,fine,tPen\WObj:=wPaper;
    MoveL Offs(pOrigin,154.10,127.79,6.00),v60,z5,tPen\WObj:=wPaper;
    MoveL Offs(pOrigin,173.13,126.68,6.00),vTravel,z5,tPen\WObj:=wPaper;
    MoveL Offs(pOrigin,173.13,126.68,0.00),v60,z0,tPen\WObj:=wPaper;
    MoveL Offs(pOrigin,199.86,99.95,0.00),v40,z0,tPen\WObj:=wPaper;
    MoveL Offs(pOrigin,199.17,100.26,0.00),v40,z0,tPen\WObj:=wPaper;
    MoveL Offs(pOrigin,192.06,93.16,0.00),v40,z0,tPen\WObj:=wPaper;
    MoveL Offs(pOrigin,192.61,92.27,0.00),v40,z0,tPen\WObj:=wPaper;
    MoveL Offs(pOrigin,173.20,111.68,0.00),v40,z0,tPen\WObj:=wPaper;
    MoveL Offs(pOrigin,174.24,111.18,0.00),v40,z0,tPen\WObj:=wPaper;
    MoveL Offs(pOrigin,196.31,133.25,0.00),v40,z0,tPen\WObj:=wPaper;
    MoveL Offs(pOrigin,195.70,133.97,0.00),v40,z0,tPen\WObj:=wPaper;
    MoveL Offs(pOrigin,200.16,129.52,0.00),v40,z0,tPen\WObj:=wPaper;
    MoveL Offs(pOrigin,199.40,128.88,0.00),v40,z0,tPen\WObj:=wPaper;
    MoveL Offs(pOrigin,174.16,103.63,0.00),v40,z0,tPen\WObj:=wPaper;
    MoveL Offs(pOrigin,175.10,103.35,0.00),v40,z0,tPen\WObj:=wPaper;
    MoveL Offs(pOrigin,198.50,103.35,0.00),v40,z0,tPen\WObj:=wPaper;
    MoveL Offs(pOrigin,199.16,103.24,0.00),v40,z0,tPen\WObj:=wPaper;
    MoveL Offs(pOrigin,189.08,93.17,0.00),v40,z0,tPen\WObj:=wPaper;
    MoveL Offs(pOrigin,189.63,92.26,0.00),v40,z0,tPen\WObj:=wPaper;
    MoveL Offs(pOrigin,173.51,108.38,0.00),v40,z0,tPen\WObj:=wPaper;
    MoveL Offs(pOrigin,174.25,108.21,0.00),v40,z0,tPen\WObj:=wPaper;
    MoveL Offs(pOrigin,199.07,133.02,0.00),v40,z0,tPen\WObj:=wPaper;
    MoveL Offs(pOrigin,199.35,133.07,0.00),v40,z0,tPen\WObj:=wPaper;
    MoveL Offs(pOrigin,174.95,133.27,0.00),v40,z0,tPen\WObj:=wPaper;
    MoveL Offs(pOrigin,174.40,132.98,0.00),v40,z0,tPen\WObj:=wPaper;
    MoveL Offs(pOrigin,174.50,92.97,0.00),v40,z0,tPen\WObj:=wPaper;
    MoveL Offs(pOrigin,199.35,93.07,0.00),v40,z0,tPen\WObj:=wPaper;
    MoveL Offs(pOrigin,199.35,133.07,0.00),v40,z0,tPen\WObj:=wPaper;
    MoveL Offs(pOrigin,199.50,131.96,0.00),v40,z0,tPen\WObj:=wPaper;
    MoveL Offs(pOrigin,174.26,106.72,0.00),v40,z0,tPen\WObj:=wPaper;
    MoveL Offs(pOrigin,173.50,106.89,0.00),v40,z0,tPen\WObj:=wPaper;
    MoveL Offs(pOrigin,188.14,92.26,0.00),v40,z0,tPen\WObj:=wPaper;
    MoveL Offs(pOrigin,187.38,92.96,0.00),v40,z0,tPen\WObj:=wPaper;
    MoveL Offs(pOrigin,199.15,104.73,0.00),v40,z0,tPen\WObj:=wPaper;
    MoveL Offs(pOrigin,198.50,104.41,0.00),v40,z0,tPen\WObj:=wPaper;
    MoveL Offs(pOrigin,175.10,104.41,0.00),v40,z0,tPen\WObj:=wPaper;
    MoveL Offs(pOrigin,175.10,105.46,0.00),v40,z0,tPen\WObj:=wPaper;
    MoveL Offs(pOrigin,198.50,105.46,0.00),v40,z0,tPen\WObj:=wPaper;
    MoveL Offs(pOrigin,199.15,106.22,0.00),v40,z0,tPen\WObj:=wPaper;
    MoveL Offs(pOrigin,185.89,92.96,0.00),v40,fine,tPen\WObj:=wPaper;
    MoveL Offs(pOrigin,185.89,92.96,6.00),v60,z5,tPen\WObj:=wPaper;
    MoveL Offs(pOrigin,186.86,92.04,6.00),vTravel,z5,tPen\WObj:=wPaper;
    MoveL Offs(pOrigin,186.86,92.04,0.00),v60,z0,tPen\WObj:=wPaper;
    MoveL Offs(pOrigin,173.29,105.62,0.00),v40,z0,tPen\WObj:=wPaper;
    MoveL Offs(pOrigin,174.26,105.23,0.00),v40,z0,tPen\WObj:=wPaper;
    MoveL Offs(pOrigin,199.40,130.36,0.00),v40,z0,tPen\WObj:=wPaper;
    MoveL Offs(pOrigin,198.65,130.81,0.00),v40,z0,tPen\WObj:=wPaper;
    MoveL Offs(pOrigin,175.10,130.81,0.00),v40,z0,tPen\WObj:=wPaper;
    MoveL Offs(pOrigin,174.30,130.65,0.00),v40,z0,tPen\WObj:=wPaper;
    MoveL Offs(pOrigin,176.95,133.30,0.00),v40,z0,tPen\WObj:=wPaper;
    MoveL Offs(pOrigin,176.34,133.92,0.00),v40,z0,tPen\WObj:=wPaper;
    MoveL Offs(pOrigin,199.79,110.48,0.00),v40,z0,tPen\WObj:=wPaper;
    MoveL Offs(pOrigin,199.24,110.79,0.00),v40,z0,tPen\WObj:=wPaper;
    MoveL Offs(pOrigin,181.32,92.87,0.00),v40,z0,tPen\WObj:=wPaper;
    MoveL Offs(pOrigin,180.91,92.02,0.00),v40,z0,tPen\WObj:=wPaper;
    MoveL Offs(pOrigin,173.37,99.55,0.00),v40,z0,tPen\WObj:=wPaper;
    MoveL Offs(pOrigin,174.17,99.16,0.00),v40,z0,tPen\WObj:=wPaper;
    MoveL Offs(pOrigin,199.42,124.41,0.00),v40,z0,tPen\WObj:=wPaper;
    MoveL Offs(pOrigin,199.93,123.78,0.00),v40,z0,tPen\WObj:=wPaper;
    MoveL Offs(pOrigin,189.75,133.96,0.00),v40,z0,tPen\WObj:=wPaper;
    MoveL Offs(pOrigin,190.46,133.37,0.00),v40,z0,tPen\WObj:=wPaper;
    MoveL Offs(pOrigin,174.23,117.14,0.00),v40,z0,tPen\WObj:=wPaper;
    MoveL Offs(pOrigin,175.25,117.08,0.00),v40,z0,tPen\WObj:=wPaper;
    MoveL Offs(pOrigin,198.35,117.08,0.00),v40,z0,tPen\WObj:=wPaper;
    MoveL Offs(pOrigin,199.12,116.64,0.00),v40,z0,tPen\WObj:=wPaper;
    MoveL Offs(pOrigin,175.36,92.88,0.00),v40,z0,tPen\WObj:=wPaper;
    MoveL Offs(pOrigin,174.63,92.32,0.00),v40,z0,tPen\WObj:=wPaper;
    MoveL Offs(pOrigin,173.68,93.28,0.00),v40,z0,tPen\WObj:=wPaper;
    MoveL Offs(pOrigin,174.40,93.42,0.00),v40,z0,tPen\WObj:=wPaper;
    MoveL Offs(pOrigin,199.22,118.24,0.00),v40,z0,tPen\WObj:=wPaper;
  ENDPROC

